REGION Network 7: flowrate ratio difference
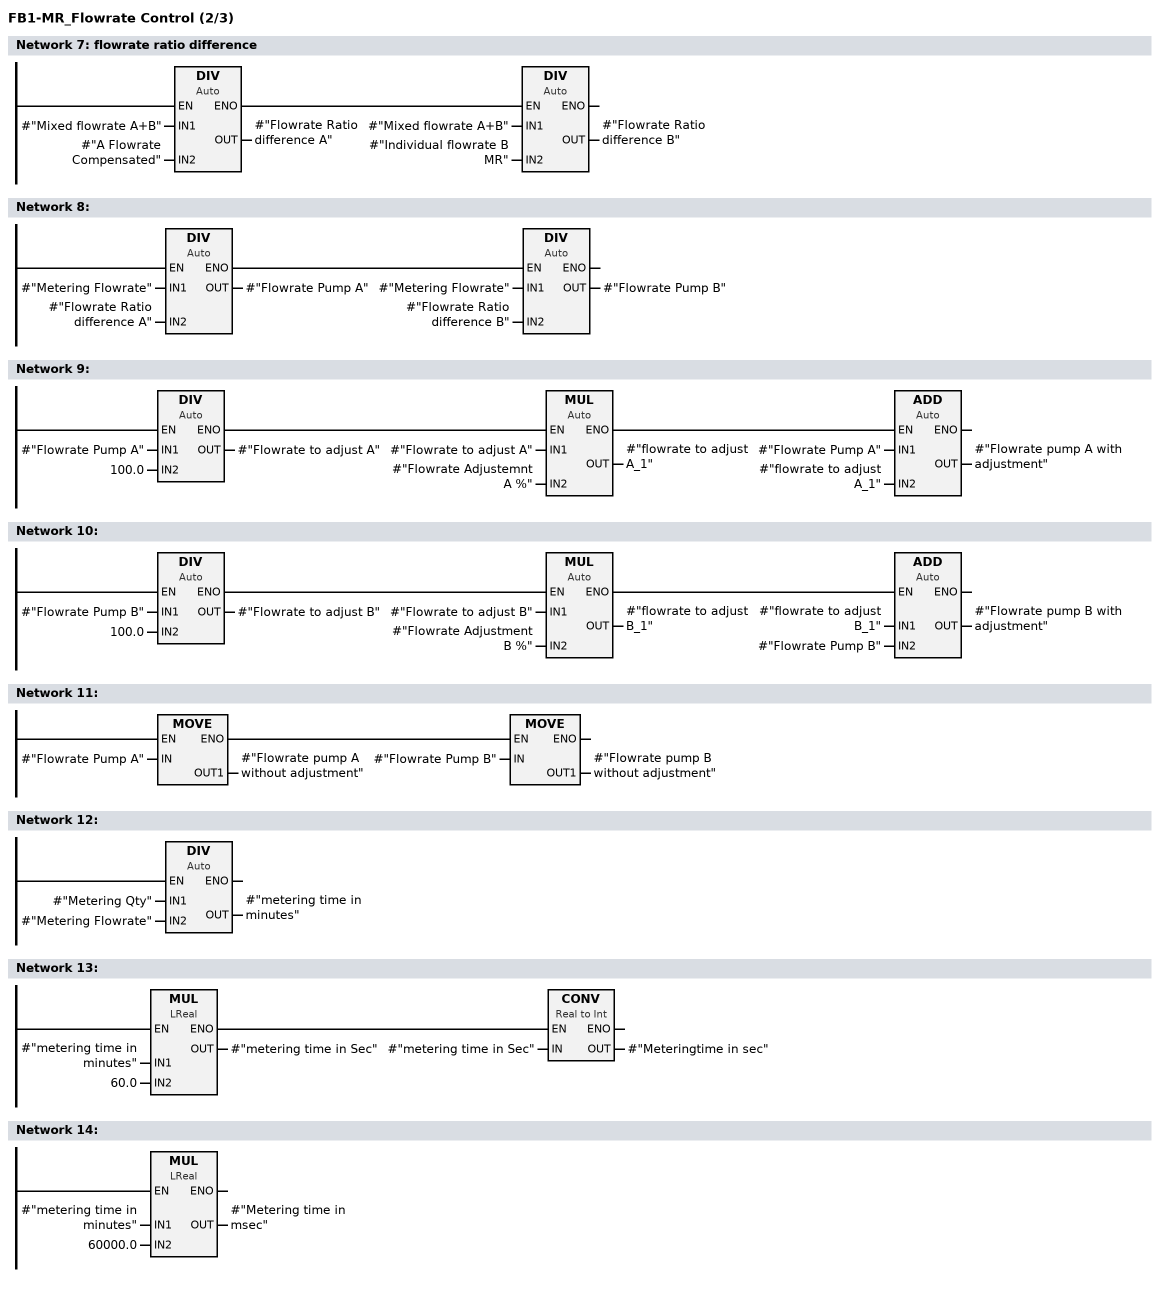
   RUNG wire#powerrail
      Div(in1 := #"Mixed flowrate A+B", in2 := #"A Flowrate Compensated", out => #"Flowrate Ratio difference A")
      Div(in1 := #"Mixed flowrate A+B", in2 := #"Individual flowrate B MR", out => #"Flowrate Ratio difference B")
   END_RUNG
   // the same network as SCL:
   #"Flowrate Ratio difference A" := #"Mixed flowrate A+B" / #"A Flowrate Compensated";
   #"Flowrate Ratio difference B" := #"Mixed flowrate A+B" / #"Individual flowrate B MR";
END_REGION

REGION Network 8
   RUNG wire#powerrail
      Div(in1 := #"Metering Flowrate", in2 := #"Flowrate Ratio difference A", out => #"Flowrate Pump A")
      Div(in1 := #"Metering Flowrate", in2 := #"Flowrate Ratio difference B", out => #"Flowrate Pump B")
   END_RUNG
   // the same network as SCL:
   #"Flowrate Pump A" := #"Metering Flowrate" / #"Flowrate Ratio difference A";
   #"Flowrate Pump B" := #"Metering Flowrate" / #"Flowrate Ratio difference B";
END_REGION

REGION Network 9
   RUNG wire#powerrail
      Div(in1 := #"Flowrate Pump A", in2 := 100.0, out => #"Flowrate to adjust A")
      Mul(in1 := #"Flowrate to adjust A", in2 := #"Flowrate Adjustemnt A %", out => #"flowrate to adjust A_1")
      Add(in1 := #"Flowrate Pump A", in2 := #"flowrate to adjust A_1", out => #"Flowrate pump A with adjustment")
   END_RUNG
   // the same network as SCL:
   #"Flowrate to adjust A" := #"Flowrate Pump A" / 100.0;
   #"flowrate to adjust A_1" := #"Flowrate to adjust A" * #"Flowrate Adjustemnt A %";
   #"Flowrate pump A with adjustment" := #"Flowrate Pump A" + #"flowrate to adjust A_1";
END_REGION

REGION Network 10
   RUNG wire#powerrail
      Div(in1 := #"Flowrate Pump B", in2 := 100.0, out => #"Flowrate to adjust B")
      Mul(in1 := #"Flowrate to adjust B", in2 := #"Flowrate Adjustment B %", out => #"flowrate to adjust B_1")
      Add(in1 := #"flowrate to adjust B_1", in2 := #"Flowrate Pump B", out => #"Flowrate pump B with adjustment")
   END_RUNG
   // the same network as SCL:
   #"Flowrate to adjust B" := #"Flowrate Pump B" / 100.0;
   #"flowrate to adjust B_1" := #"Flowrate to adjust B" * #"Flowrate Adjustment B %";
   #"Flowrate pump B with adjustment" := #"flowrate to adjust B_1" + #"Flowrate Pump B";
END_REGION

REGION Network 11
   RUNG wire#powerrail
      Move(in := #"Flowrate Pump A", out1 => #"Flowrate pump A without adjustment")
      Move(in := #"Flowrate Pump B", out1 => #"Flowrate pump B without adjustment")
   END_RUNG
   // the same network as SCL:
   #"Flowrate pump A without adjustment" := #"Flowrate Pump A";
   #"Flowrate pump B without adjustment" := #"Flowrate Pump B";
END_REGION

REGION Network 12
   RUNG wire#powerrail
      Div(in1 := #"Metering Qty", in2 := #"Metering Flowrate", out => #"metering time in minutes")
   END_RUNG
   // the same network as SCL:
   #"metering time in minutes" := #"Metering Qty" / #"Metering Flowrate";
END_REGION

REGION Network 13
   RUNG wire#powerrail
      { S7_Templates := "SrcType := LReal" } Mul(in1 := #"metering time in minutes", in2 := 60.0, out => #"metering time in Sec")
      { S7_Templates := "[SrcType := Real, DestType := Int]" } Convert(in := #"metering time in Sec", out => #"Meteringtime in sec")
   END_RUNG
   // the same network as SCL:
   #"metering time in Sec" := #"metering time in minutes" * 60.0;
   #"Meteringtime in sec" := REAL_TO_INT(#"metering time in Sec");
END_REGION

REGION Network 14
   RUNG wire#powerrail
      { S7_Templates := "SrcType := LReal" } Mul(in1 := #"metering time in minutes", in2 := 60000.0, out => #"Metering time in msec")
   END_RUNG
   // the same network as SCL:
   #"Metering time in msec" := #"metering time in minutes" * 60000.0;
END_REGION

REGION Network 15
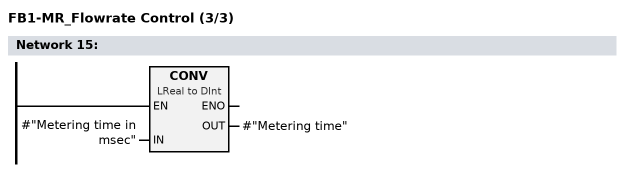
   RUNG wire#powerrail
      { S7_Templates := "[SrcType := LReal, DestType := DInt]" } Convert(in := #"Metering time in msec", out => #"Metering time")
   END_RUNG
   // the same network as SCL:
   #"Metering time" := LREAL_TO_DINT(#"Metering time in msec");
END_REGION
END_FUNCTION_BLOCK

ORGANIZATION_BLOCK "Startup"   // OB100, LAD, Startup
TITLE = "Complete Restart"
{ S7_Optimized_Access := 'TRUE' }
VERSION : 0.1
// stored: AutoNumber true, IsIECCheckEnabled false, SetENOAutomatically false
   VAR_INPUT
      LostRetentive : Bool;   // True if retentive data are lost
      LostRTC : Bool;   // True if date and time are lost
   END_VAR
BEGIN

REGION Network 1
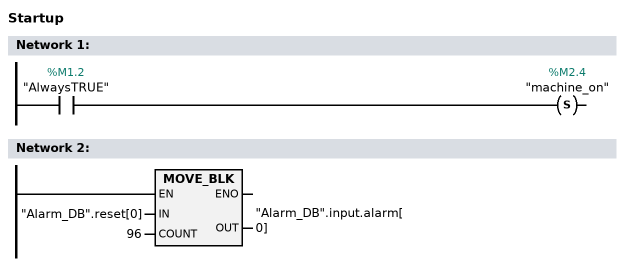
   RUNG wire#powerrail
      Contact( "AlwaysTRUE" )
      S_Coil( "machine_on" )
   END_RUNG
   // the same network as SCL:
   IF "AlwaysTRUE" THEN "machine_on" := TRUE; END_IF;
END_REGION

REGION Network 2
   MOVE_BLK(IN := "Alarm_DB".reset[0], COUNT := 96, OUT => "Alarm_DB".input.alarm[0]);
END_REGION
END_ORGANIZATION_BLOCK

FUNCTION "Alram_Scroll" : Void   // FC15, LAD
{ S7_Optimized_Access := 'TRUE' }
VERSION : 0.1
// stored: AutoNumber true, IsIECCheckEnabled false, SetENOAutomatically false, UDAEnableTagReadback false
   VAR CONSTANT
      "AlramDisplay time" : DInt := 2000;
   END_VAR
BEGIN

REGION Network 1
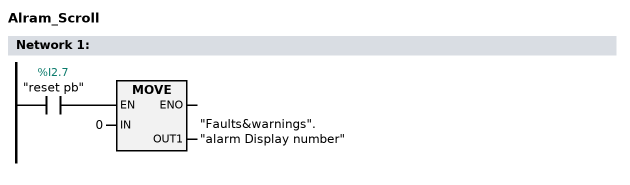
   RUNG wire#powerrail
      Contact( "reset pb" )
      Move(in := 0, out1 => "Faults&warnings"."alarm Display number")
   END_RUNG
   // the same network as SCL:
   IF "reset pb" THEN "Faults&warnings"."alarm Display number" := 0; END_IF;
END_REGION
END_FUNCTION

FUNCTION_BLOCK "FB10-Condition Check"   // FB10, LAD
{ S7_Optimized_Access := 'TRUE' }
VERSION : 0.1
// stored: AutoNumber false, IsIECCheckEnabled false, IsRetainMemResEnabled false, MemoryReserve 100, SetENOAutomatically false, UDAEnableTagReadback false
   VAR_INPUT
      "Time" : DInt;
      "Pump ON delay" : DInt;
      Check_Time { ExternalAccessible := 'False'; ExternalVisible := 'False'; ExternalWritable := 'False'} : DInt;
      Pressure_SP { ExternalAccessible := 'False'; ExternalVisible := 'False'; ExternalWritable := 'False'} : Real;
      Pressure_tolerance { ExternalAccessible := 'False'; ExternalVisible := 'False'; ExternalWritable := 'False'} : Real;
      Current_pressure { ExternalAccessible := 'False'; ExternalVisible := 'False'; ExternalWritable := 'False'} : Real;
      selected { ExternalAccessible := 'False'; ExternalVisible := 'False'; ExternalWritable := 'False'} : Bool;
   END_VAR
   VAR_OUTPUT
      "dispensing Time PV" : Int;
      "Checking Time pv" { ExternalAccessible := 'False'; ExternalVisible := 'False'; ExternalWritable := 'False'} : Int;
      test_ok { ExternalAccessible := 'False'; ExternalVisible := 'False'; ExternalWritable := 'False'} : Bool;
      test_nok { ExternalAccessible := 'False'; ExternalVisible := 'False'; ExternalWritable := 'False'} : Bool;
      test_fail { ExternalAccessible := 'False'; ExternalVisible := 'False'; ExternalWritable := 'False'} : Bool;
   END_VAR
   VAR_IN_OUT
      "Start ConditonCheck" : Bool;
      "Stop ConditonCheck" : Bool;
      "ConditonCheck Running" : Bool;
      "ConditonCheck completed" : Bool;
      "ON Gear Pump" : Bool;
      "ON inlet" : Bool;
   END_VAR
   VAR
      "dispensing time done" : Bool;
      "dispensing time in sec" : DInt;
      "timer in sec" : DInt;
      "timer PV in sec" : DInt;
      "timer input" : DInt;
      IEC_Timer_0_Instance { S7_SetPoint := 'True'} : TON_TIME;
      IEC_Timer_0_Instance_1 { S7_SetPoint := 'True'} : TON_TIME;
      IEC_Timer_0_Instance_2 { S7_SetPoint := 'True'} : TON_TIME;
      IEC_Timer_0_Instance_4 { S7_SetPoint := 'True'} : TON_TIME;
      "Press+ve" { ExternalAccessible := 'False'; ExternalVisible := 'False'; ExternalWritable := 'False'; S7_SetPoint := 'True'} : Real;
      "Press-ve" { ExternalAccessible := 'False'; ExternalVisible := 'False'; ExternalWritable := 'False'} : Real;
      IEC_Timer_0_Instance_3 { ExternalAccessible := 'False'; ExternalVisible := 'False'; ExternalWritable := 'False'; S7_SetPoint := 'True'} : TON_TIME;
      Checktime_ms { ExternalAccessible := 'False'; ExternalVisible := 'False'; ExternalWritable := 'False'; S7_SetPoint := 'True'} : DInt;
      Check_timesec { ExternalAccessible := 'False'; ExternalVisible := 'False'; ExternalWritable := 'False'} : DInt;
      temp_ons { ExternalAccessible := 'False'; ExternalVisible := 'False'; ExternalWritable := 'False'} : Bool;
   END_VAR
   VAR_TEMP   // added for the SCL form of the ladder/FBD networks
      _w1 : Bool;
   END_VAR
BEGIN

REGION Network 1
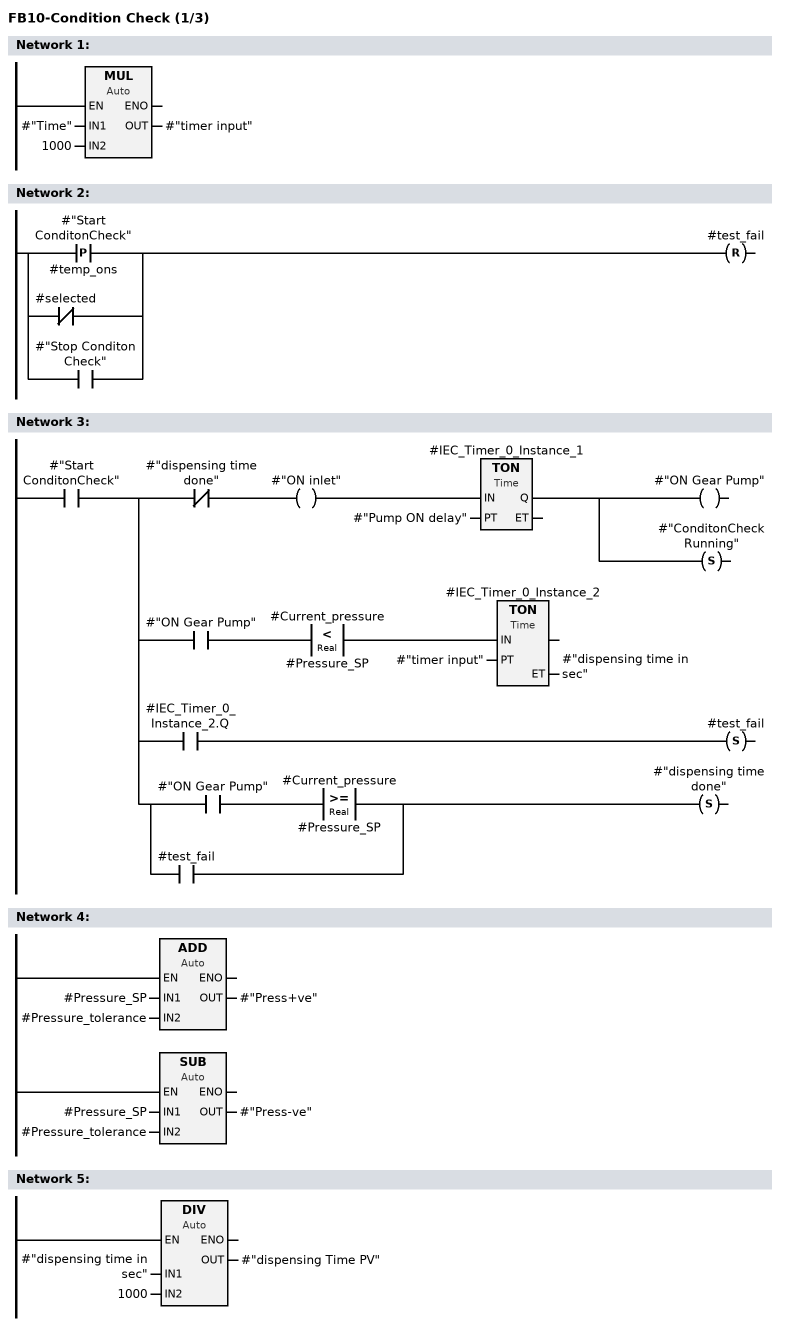
   RUNG wire#powerrail
      Mul(in1 := #"Time", in2 := 1000, out => #"timer input")
   END_RUNG
   // the same network as SCL:
   #"timer input" := #"Time" * 1000;
END_REGION

REGION Network 2
   RUNG wire#powerrail
      P_Contact(operand := #"Start ConditonCheck", bit := #temp_ons)
      wire#w1
      R_Coil( #test_fail )
   END_RUNG
   RUNG wire#powerrail
      I_Contact( #selected )
   END_RUNG wire#w1
   RUNG wire#powerrail
      Contact( #"Stop ConditonCheck" )
   END_RUNG wire#w1
   // the same network as SCL:
   #_w1 := #"Start ConditonCheck" AND NOT #temp_ons;   // rising edge of #"Start ConditonCheck"
   #temp_ons := #"Start ConditonCheck";
   IF #_w1 OR NOT #selected OR #"Stop ConditonCheck" THEN #test_fail := FALSE; END_IF;
END_REGION

REGION Network 3
   RUNG wire#powerrail
      Contact( #"Start ConditonCheck" )
      wire#w1
      I_Contact( #"dispensing time done" )
      Coil( #"ON inlet" )
      { S7_Templates := "time_type := Time" } #IEC_Timer_0_Instance_1.TON(pt := #"Pump ON delay", et =>)
      wire#w2
      Coil( #"ON Gear Pump" )
   END_RUNG
   RUNG wire#w2
      S_Coil( #"ConditonCheck Running" )
   END_RUNG
   RUNG wire#w1
      Contact( #"ON Gear Pump" )
      { S7_Templates := "SrcType := Real" } LT_Contact(in1 := #Current_pressure, in2 := #Pressure_SP)
      { S7_Templates := "time_type := Time" } #IEC_Timer_0_Instance_2.TON(pt := #"timer input", et => #"dispensing time in sec")
   END_RUNG
   RUNG wire#w1
      Contact( #IEC_Timer_0_Instance_2.Q )
      S_Coil( #test_fail )
   END_RUNG
   RUNG wire#w1
      Contact( #"ON Gear Pump" )
      { S7_Templates := "SrcType := Real" } GE_Contact(in1 := #Current_pressure, in2 := #Pressure_SP)
      wire#w3
      S_Coil( #"dispensing time done" )
   END_RUNG
   RUNG wire#w1
      Contact( #test_fail )
   END_RUNG wire#w3
   // the same network as SCL:
   #"ON inlet" := #"Start ConditonCheck" AND NOT #"dispensing time done";
   #IEC_Timer_0_Instance_1(IN := #"ON inlet", PT := #"Pump ON delay");   // TON
   #"ON Gear Pump" := #IEC_Timer_0_Instance_1.Q;
   IF #IEC_Timer_0_Instance_1.Q THEN #"ConditonCheck Running" := TRUE; END_IF;
   #IEC_Timer_0_Instance_2(IN := #"Start ConditonCheck" AND #"ON Gear Pump" AND (#Current_pressure < #Pressure_SP),   // TON
                           PT := #"timer input",
                           ET => #"dispensing time in sec");
   IF #"Start ConditonCheck" AND #IEC_Timer_0_Instance_2.Q THEN #test_fail := TRUE; END_IF;
   IF #"Start ConditonCheck" AND ((#"ON Gear Pump" AND (#Current_pressure >= #Pressure_SP)) OR #test_fail) THEN
       #"dispensing time done" := TRUE;
   END_IF;
END_REGION

REGION Network 4
   RUNG wire#powerrail
      Add(in1 := #Pressure_SP, in2 := #Pressure_tolerance, out => #"Press+ve")
   END_RUNG
   RUNG wire#powerrail
      Sub(in1 := #Pressure_SP, in2 := #Pressure_tolerance, out => #"Press-ve")
   END_RUNG
   // the same network as SCL:
   #"Press+ve" := #Pressure_SP + #Pressure_tolerance;
   #"Press-ve" := #Pressure_SP - #Pressure_tolerance;
END_REGION

REGION Network 5
   RUNG wire#powerrail
      Div(in1 := #"dispensing time in sec", in2 := 1000, out => #"dispensing Time PV")
   END_RUNG
   // the same network as SCL:
   #"dispensing Time PV" := #"dispensing time in sec" / 1000;
END_REGION

REGION Network 6
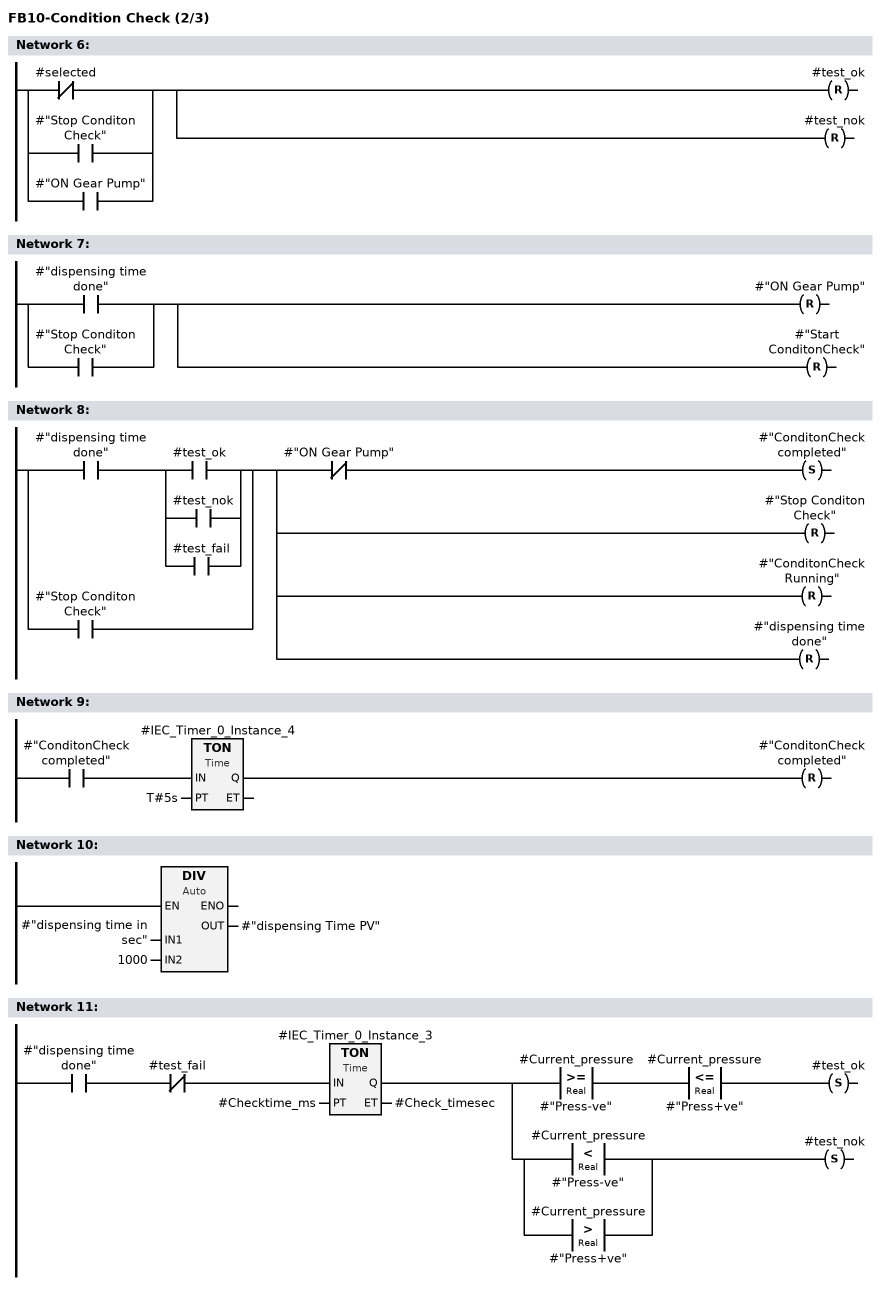
   RUNG wire#powerrail
      I_Contact( #selected )
      wire#w1
      R_Coil( #test_ok )
   END_RUNG
   RUNG wire#powerrail
      Contact( #"Stop ConditonCheck" )
   END_RUNG wire#w1
   RUNG wire#powerrail
      Contact( #"ON Gear Pump" )
   END_RUNG wire#w1
   RUNG wire#w1
      R_Coil( #test_nok )
   END_RUNG
   // the same network as SCL:
   IF NOT #selected OR #"Stop ConditonCheck" OR #"ON Gear Pump" THEN
       #test_ok := FALSE;
       #test_nok := FALSE;
   END_IF;
END_REGION

REGION Network 7
   RUNG wire#powerrail
      Contact( #"dispensing time done" )
      wire#w1
      R_Coil( #"ON Gear Pump" )
   END_RUNG
   RUNG wire#powerrail
      Contact( #"Stop ConditonCheck" )
   END_RUNG wire#w1
   RUNG wire#w1
      R_Coil( #"Start ConditonCheck" )
   END_RUNG
   // the same network as SCL:
   IF #"dispensing time done" OR #"Stop ConditonCheck" THEN
       #"ON Gear Pump" := FALSE;
       #"Start ConditonCheck" := FALSE;
   END_IF;
END_REGION

REGION Network 8
   RUNG wire#powerrail
      Contact( #"dispensing time done" )
      wire#w1
      Contact( #test_ok )
      wire#w2
      I_Contact( #"ON Gear Pump" )
      S_Coil( #"ConditonCheck completed" )
   END_RUNG
   RUNG wire#w1
      Contact( #test_nok )
   END_RUNG wire#w2
   RUNG wire#w1
      Contact( #test_fail )
   END_RUNG wire#w2
   RUNG wire#powerrail
      Contact( #"Stop ConditonCheck" )
   END_RUNG wire#w2
   RUNG wire#w2
      R_Coil( #"Stop ConditonCheck" )
   END_RUNG
   RUNG wire#w2
      R_Coil( #"ConditonCheck Running" )
   END_RUNG
   RUNG wire#w2
      R_Coil( #"dispensing time done" )
   END_RUNG
   // the same network as SCL:
   #_w1 := (#"dispensing time done" AND (#test_ok OR #test_nok OR #test_fail)) OR #"Stop ConditonCheck";
   IF #_w1 AND NOT #"ON Gear Pump" THEN #"ConditonCheck completed" := TRUE; END_IF;
   IF #_w1 THEN
       #"Stop ConditonCheck" := FALSE;
       #"ConditonCheck Running" := FALSE;
       #"dispensing time done" := FALSE;
   END_IF;
END_REGION

REGION Network 9
   RUNG wire#powerrail
      Contact( #"ConditonCheck completed" )
      { S7_Templates := "time_type := Time" } #IEC_Timer_0_Instance_4.TON(pt := T#5s, et =>)
      R_Coil( #"ConditonCheck completed" )
   END_RUNG
   // the same network as SCL:
   #IEC_Timer_0_Instance_4(IN := #"ConditonCheck completed", PT := T#5s);   // TON
   IF #IEC_Timer_0_Instance_4.Q THEN #"ConditonCheck completed" := FALSE; END_IF;
END_REGION

REGION Network 10
   RUNG wire#powerrail
      Div(in1 := #"dispensing time in sec", in2 := 1000, out => #"dispensing Time PV")
   END_RUNG
   // the same network as SCL:
   #"dispensing Time PV" := #"dispensing time in sec" / 1000;
END_REGION

REGION Network 11
   RUNG wire#powerrail
      Contact( #"dispensing time done" )
      I_Contact( #test_fail )
      { S7_Templates := "time_type := Time" } #IEC_Timer_0_Instance_3.TON(pt := #Checktime_ms, et => #Check_timesec)
      wire#w1
      { S7_Templates := "SrcType := Real" } GE_Contact(in1 := #Current_pressure, in2 := #"Press-ve")
      { S7_Templates := "SrcType := Real" } LE_Contact(in1 := #Current_pressure, in2 := #"Press+ve")
      S_Coil( #test_ok )
   END_RUNG
   RUNG wire#w1
      { S7_Templates := "SrcType := Real" } LT_Contact(in1 := #Current_pressure, in2 := #"Press-ve")
      wire#w2
      S_Coil( #test_nok )
   END_RUNG
   RUNG wire#w1
      { S7_Templates := "SrcType := Real" } GT_Contact(in1 := #Current_pressure, in2 := #"Press+ve")
   END_RUNG wire#w2
   // the same network as SCL:
   #IEC_Timer_0_Instance_3(IN := #"dispensing time done" AND NOT #test_fail,   // TON
                           PT := #Checktime_ms,
                           ET => #Check_timesec);
   IF #IEC_Timer_0_Instance_3.Q AND (#Current_pressure >= #"Press-ve") AND (#Current_pressure <= #"Press+ve") THEN
       #test_ok := TRUE;
   END_IF;
   IF #IEC_Timer_0_Instance_3.Q AND ((#Current_pressure < #"Press-ve") OR (#Current_pressure > #"Press+ve")) THEN
       #test_nok := TRUE;
   END_IF;
END_REGION

REGION Network 12
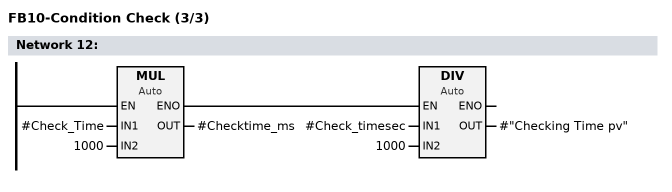
   RUNG wire#powerrail
      Mul(in1 := #Check_Time, in2 := 1000, out => #Checktime_ms)
      Div(in1 := #Check_timesec, in2 := 1000, out => #"Checking Time pv")
   END_RUNG
   // the same network as SCL:
   #Checktime_ms := #Check_Time * 1000;
   #"Checking Time pv" := #Check_timesec / 1000;
END_REGION
END_FUNCTION_BLOCK

FUNCTION_BLOCK "MixingRatio"   // FB11, LAD
{ S7_Optimized_Access := 'TRUE' }
VERSION : 0.1
// stored: AutoNumber true, IsIECCheckEnabled false, IsRetainMemResEnabled false, MemoryReserve 100, SetENOAutomatically false, UDAEnableTagReadback false
   VAR_INPUT
      "Pump size A in ml" : Real;
      "Pump size B in ml" : Real;
      "Pump speed A_Max" : Real;
      "Pump speed B_Max" : Real;
      "Pump speed A_Passive" : Real;
      "Pump speed B_Passive" : Real;
      "Mixing ratio A100:B" : Real;
      "No.of Component" : Int;
      "Density A" : Real;
      "Density B" : Real;
      "Mixed Flowrate Set" : Real;
      "Flowrate Type" : Int;
   END_VAR
   VAR_OUTPUT
      "Maximum Flowrate A" : Real;
      "Maximum Flowrate B" : Real;
      "Maximum Flowrate A_Limited" : Real;
      "Maximum Flowrate B_Limited" : Real;
      "Maximum Flowrate Mixed" : Real;
      "Required flowrate A" : Real;
      "Required flowrate B" : Real;
   END_VAR
   VAR
      "Pump size A actual" : Real;
      "Pump size B actual" : Real;
      "Max flowrate A" : Real;
      "Max flowrate B" : Real;
      "Ratio margin B" : Real;
      "usable A flowrate per B ratio" : Real;
      "maximum mixed flowrate" : Real;
      "usable flowrate A per ratio" : Real;
      "usable flowrate B per ratio" : Real;
      "Flowrate difference A" : Real;
      "Flowrate difference B" : Real;
      "target flowrate A" : Real;
      "target flowrate B" : Real;
   END_VAR
   VAR_TEMP   // added for the SCL form of the ladder/FBD networks
      _w1 : Bool;
   END_VAR
BEGIN

REGION Network 1
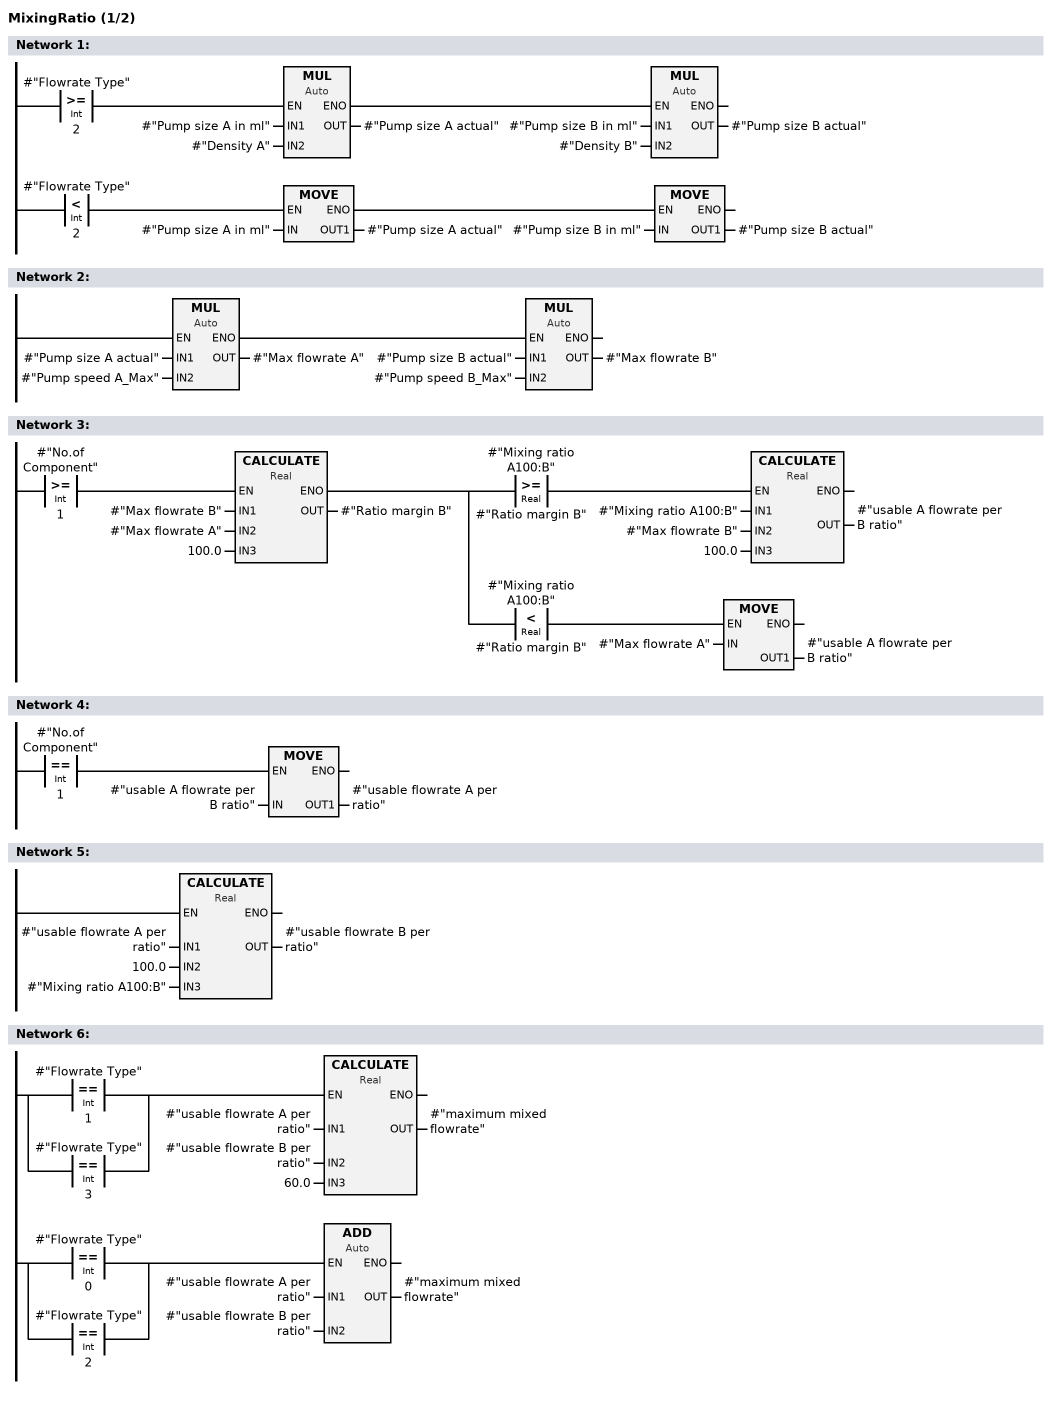
   RUNG wire#powerrail
      { S7_Templates := "SrcType := Int" } GE_Contact(in1 := #"Flowrate Type", in2 := 2)
      Mul(in1 := #"Pump size A in ml", in2 := #"Density A", out => #"Pump size A actual")
      Mul(in1 := #"Pump size B in ml", in2 := #"Density B", out => #"Pump size B actual")
   END_RUNG
   RUNG wire#powerrail
      { S7_Templates := "SrcType := Int" } LT_Contact(in1 := #"Flowrate Type", in2 := 2)
      Move(in := #"Pump size A in ml", out1 => #"Pump size A actual")
      Move(in := #"Pump size B in ml", out1 => #"Pump size B actual")
   END_RUNG
   // the same network as SCL:
   IF #"Flowrate Type" >= 2 THEN
       #"Pump size A actual" := #"Pump size A in ml" * #"Density A";
       #"Pump size B actual" := #"Pump size B in ml" * #"Density B";
   END_IF;
   IF #"Flowrate Type" < 2 THEN
       #"Pump size A actual" := #"Pump size A in ml";
       #"Pump size B actual" := #"Pump size B in ml";
   END_IF;
END_REGION

REGION Network 2
   RUNG wire#powerrail
      Mul(in1 := #"Pump size A actual", in2 := #"Pump speed A_Max", out => #"Max flowrate A")
      Mul(in1 := #"Pump size B actual", in2 := #"Pump speed B_Max", out => #"Max flowrate B")
   END_RUNG
   // the same network as SCL:
   #"Max flowrate A" := #"Pump size A actual" * #"Pump speed A_Max";
   #"Max flowrate B" := #"Pump size B actual" * #"Pump speed B_Max";
END_REGION

REGION Network 3
   RUNG wire#powerrail
      { S7_Templates := "SrcType := Int" } GE_Contact(in1 := #"No.of Component", in2 := 1)
      { S7_Templates := "SrcType := Real"; S7_Expression := "(IN1/IN2)*IN3" } Calculate(in1 := #"Max flowrate B", in2 := #"Max flowrate A", in3 := 100.0, out => #"Ratio margin B")
      wire#w1
      { S7_Templates := "SrcType := Real" } GE_Contact(in1 := #"Mixing ratio A100:B", in2 := #"Ratio margin B")
      { S7_Templates := "SrcType := Real"; S7_Expression := "IN2/(IN1/IN3)" } Calculate(in1 := #"Mixing ratio A100:B", in2 := #"Max flowrate B", in3 := 100.0, out => #"usable A flowrate per B ratio")
   END_RUNG
   RUNG wire#w1
      { S7_Templates := "SrcType := Real" } LT_Contact(in1 := #"Mixing ratio A100:B", in2 := #"Ratio margin B")
      Move(in := #"Max flowrate A", out1 => #"usable A flowrate per B ratio")
   END_RUNG
   // the same network as SCL:
   #_w1 := #"No.of Component" >= 1;
   IF #_w1 THEN #"Ratio margin B" := (#"Max flowrate B"/#"Max flowrate A")*100.0; END_IF;
   IF #_w1 AND (#"Mixing ratio A100:B" >= #"Ratio margin B") THEN
       #"usable A flowrate per B ratio" := #"Max flowrate B"/(#"Mixing ratio A100:B"/100.0);
   END_IF;
   IF #_w1 AND (#"Mixing ratio A100:B" < #"Ratio margin B") THEN
       #"usable A flowrate per B ratio" := #"Max flowrate A";
   END_IF;
END_REGION

REGION Network 4
   RUNG wire#powerrail
      { S7_Templates := "SrcType := Int" } EQ_Contact(in1 := #"No.of Component", in2 := 1)
      Move(in := #"usable A flowrate per B ratio", out1 => #"usable flowrate A per ratio")
   END_RUNG
   // the same network as SCL:
   IF #"No.of Component" = 1 THEN #"usable flowrate A per ratio" := #"usable A flowrate per B ratio"; END_IF;
END_REGION

REGION Network 5
   RUNG wire#powerrail
      { S7_Templates := "SrcType := Real"; S7_Expression := "(IN1/IN2)*IN3" } Calculate(in1 := #"usable flowrate A per ratio", in2 := 100.0, in3 := #"Mixing ratio A100:B", out => #"usable flowrate B per ratio")
   END_RUNG
   // the same network as SCL:
   #"usable flowrate B per ratio" := (#"usable flowrate A per ratio"/100.0)*#"Mixing ratio A100:B";
END_REGION

REGION Network 6
   RUNG wire#powerrail
      { S7_Templates := "SrcType := Int" } EQ_Contact(in1 := #"Flowrate Type", in2 := 1)
      wire#w1
      { S7_Templates := "SrcType := Real"; S7_Expression := "(IN1+IN2)/IN3" } Calculate(in1 := #"usable flowrate A per ratio", in2 := #"usable flowrate B per ratio", in3 := 60.0, out => #"maximum mixed flowrate")
   END_RUNG
   RUNG wire#powerrail
      { S7_Templates := "SrcType := Int" } EQ_Contact(in1 := #"Flowrate Type", in2 := 3)
   END_RUNG wire#w1
   RUNG wire#powerrail
      { S7_Templates := "SrcType := Int" } EQ_Contact(in1 := #"Flowrate Type", in2 := 0)
      wire#w2
      Add(in1 := #"usable flowrate A per ratio", in2 := #"usable flowrate B per ratio", out => #"maximum mixed flowrate")
   END_RUNG
   RUNG wire#powerrail
      { S7_Templates := "SrcType := Int" } EQ_Contact(in1 := #"Flowrate Type", in2 := 2)
   END_RUNG wire#w2
   // the same network as SCL:
   IF (#"Flowrate Type" = 1) OR (#"Flowrate Type" = 3) THEN
       #"maximum mixed flowrate" := (#"usable flowrate A per ratio"+#"usable flowrate B per ratio")/60.0;
   END_IF;
   IF (#"Flowrate Type" = 0) OR (#"Flowrate Type" = 2) THEN
       #"maximum mixed flowrate" := #"usable flowrate A per ratio" + #"usable flowrate B per ratio";
   END_IF;
END_REGION

REGION Network 7
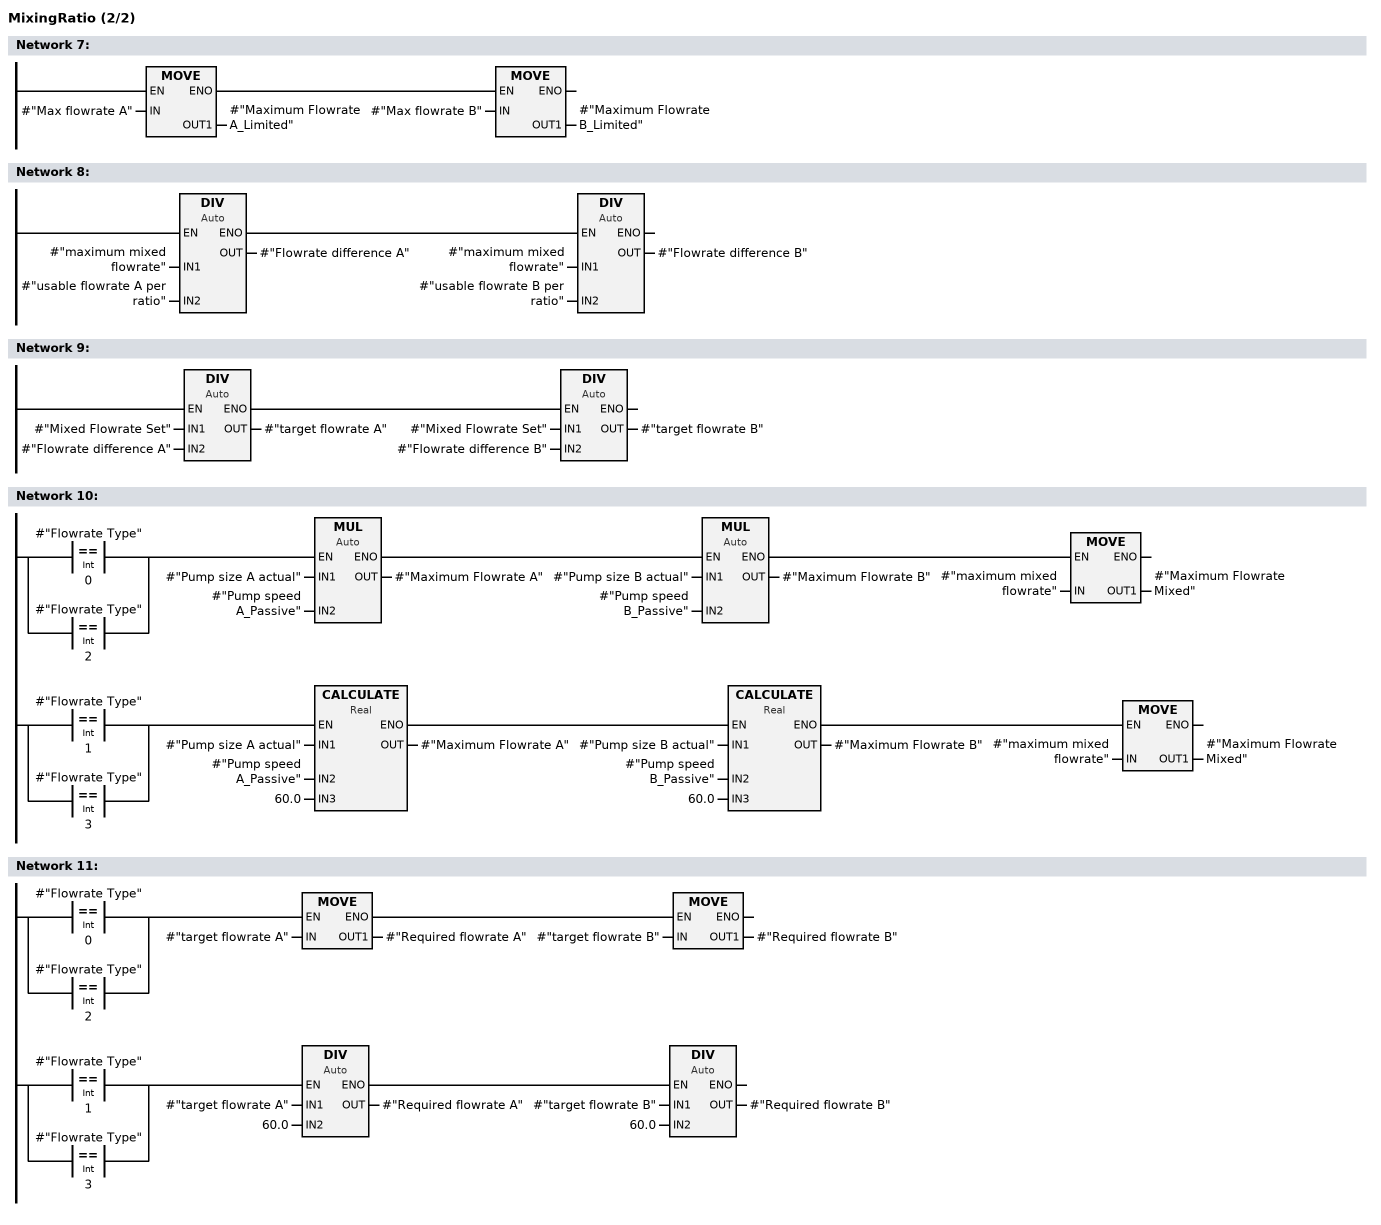
   RUNG wire#powerrail
      Move(in := #"Max flowrate A", out1 => #"Maximum Flowrate A_Limited")
      Move(in := #"Max flowrate B", out1 => #"Maximum Flowrate B_Limited")
   END_RUNG
   // the same network as SCL:
   #"Maximum Flowrate A_Limited" := #"Max flowrate A";
   #"Maximum Flowrate B_Limited" := #"Max flowrate B";
END_REGION

REGION Network 8
   RUNG wire#powerrail
      Div(in1 := #"maximum mixed flowrate", in2 := #"usable flowrate A per ratio", out => #"Flowrate difference A")
      Div(in1 := #"maximum mixed flowrate", in2 := #"usable flowrate B per ratio", out => #"Flowrate difference B")
   END_RUNG
   // the same network as SCL:
   #"Flowrate difference A" := #"maximum mixed flowrate" / #"usable flowrate A per ratio";
   #"Flowrate difference B" := #"maximum mixed flowrate" / #"usable flowrate B per ratio";
END_REGION

REGION Network 9
   RUNG wire#powerrail
      Div(in1 := #"Mixed Flowrate Set", in2 := #"Flowrate difference A", out => #"target flowrate A")
      Div(in1 := #"Mixed Flowrate Set", in2 := #"Flowrate difference B", out => #"target flowrate B")
   END_RUNG
   // the same network as SCL:
   #"target flowrate A" := #"Mixed Flowrate Set" / #"Flowrate difference A";
   #"target flowrate B" := #"Mixed Flowrate Set" / #"Flowrate difference B";
END_REGION

REGION Network 10
   RUNG wire#powerrail
      { S7_Templates := "SrcType := Int" } EQ_Contact(in1 := #"Flowrate Type", in2 := 0)
      wire#w1
      Mul(in1 := #"Pump size A actual", in2 := #"Pump speed A_Passive", out => #"Maximum Flowrate A")
      Mul(in1 := #"Pump size B actual", in2 := #"Pump speed B_Passive", out => #"Maximum Flowrate B")
      Move(in := #"maximum mixed flowrate", out1 => #"Maximum Flowrate Mixed")
   END_RUNG
   RUNG wire#powerrail
      { S7_Templates := "SrcType := Int" } EQ_Contact(in1 := #"Flowrate Type", in2 := 2)
   END_RUNG wire#w1
   RUNG wire#powerrail
      { S7_Templates := "SrcType := Int" } EQ_Contact(in1 := #"Flowrate Type", in2 := 1)
      wire#w2
      { S7_Templates := "SrcType := Real"; S7_Expression := "(IN1*IN2)/IN3" } Calculate(in1 := #"Pump size A actual", in2 := #"Pump speed A_Passive", in3 := 60.0, out => #"Maximum Flowrate A")
      { S7_Templates := "SrcType := Real"; S7_Expression := "(IN1*IN2)/IN3" } Calculate(in1 := #"Pump size B actual", in2 := #"Pump speed B_Passive", in3 := 60.0, out => #"Maximum Flowrate B")
      Move(in := #"maximum mixed flowrate", out1 => #"Maximum Flowrate Mixed")
   END_RUNG
   RUNG wire#powerrail
      { S7_Templates := "SrcType := Int" } EQ_Contact(in1 := #"Flowrate Type", in2 := 3)
   END_RUNG wire#w2
   // the same network as SCL:
   IF (#"Flowrate Type" = 0) OR (#"Flowrate Type" = 2) THEN
       #"Maximum Flowrate A" := #"Pump size A actual" * #"Pump speed A_Passive";
       #"Maximum Flowrate B" := #"Pump size B actual" * #"Pump speed B_Passive";
       #"Maximum Flowrate Mixed" := #"maximum mixed flowrate";
   END_IF;
   IF (#"Flowrate Type" = 1) OR (#"Flowrate Type" = 3) THEN
       #"Maximum Flowrate A" := (#"Pump size A actual"*#"Pump speed A_Passive")/60.0;
       #"Maximum Flowrate B" := (#"Pump size B actual"*#"Pump speed B_Passive")/60.0;
       #"Maximum Flowrate Mixed" := #"maximum mixed flowrate";
   END_IF;
END_REGION

REGION Network 11
   RUNG wire#powerrail
      { S7_Templates := "SrcType := Int" } EQ_Contact(in1 := #"Flowrate Type", in2 := 0)
      wire#w1
      Move(in := #"target flowrate A", out1 => #"Required flowrate A")
      Move(in := #"target flowrate B", out1 => #"Required flowrate B")
   END_RUNG
   RUNG wire#powerrail
      { S7_Templates := "SrcType := Int" } EQ_Contact(in1 := #"Flowrate Type", in2 := 2)
   END_RUNG wire#w1
   RUNG wire#powerrail
      { S7_Templates := "SrcType := Int" } EQ_Contact(in1 := #"Flowrate Type", in2 := 1)
      wire#w2
      Div(in1 := #"target flowrate A", in2 := 60.0, out => #"Required flowrate A")
      Div(in1 := #"target flowrate B", in2 := 60.0, out => #"Required flowrate B")
   END_RUNG
   RUNG wire#powerrail
      { S7_Templates := "SrcType := Int" } EQ_Contact(in1 := #"Flowrate Type", in2 := 3)
   END_RUNG wire#w2
   // the same network as SCL:
   IF (#"Flowrate Type" = 0) OR (#"Flowrate Type" = 2) THEN
       #"Required flowrate A" := #"target flowrate A";
       #"Required flowrate B" := #"target flowrate B";
   END_IF;
   IF (#"Flowrate Type" = 1) OR (#"Flowrate Type" = 3) THEN
       #"Required flowrate A" := #"target flowrate A" / 60.0;
       #"Required flowrate B" := #"target flowrate B" / 60.0;
   END_IF;
END_REGION
END_FUNCTION_BLOCK

FUNCTION "selection_Machine" : Void   // FC1, LAD
{ S7_Optimized_Access := 'TRUE' }
VERSION : 0.1
// stored: AutoNumber true, IsIECCheckEnabled false, SetENOAutomatically false, UDAEnableTagReadback false
BEGIN

REGION Network 1 (SCL)
   IF "selection_machie_db"."1k_2k" = TRUE THEN
       "Mixing ratio"."Mixing ratio set" := 0;
   END_IF;
END_REGION
END_FUNCTION

DATA_BLOCK "FB0-MR_Quantity Control_1_DB"   // DB24
VERSION : 0.1
// stored: AutoNumber true, DBAccessibleFromOPCUA true, InstanceOfName FB0-MR_Quantity Control_1, InstanceOfType FB
"FB0-MR_Quantity Control_1"
BEGIN
END_DATA_BLOCK

DATA_BLOCK "FB1-MR_Flowrate Control_DB"   // DB39
VERSION : 0.1
// stored: AutoNumber true, DBAccessibleFromOPCUA true, InstanceOfName FB1-MR_Flowrate Control, InstanceOfType FB
"FB1-MR_Flowrate Control"
BEGIN
END_DATA_BLOCK

DATA_BLOCK "FB10-Condition CheckA_DB"   // DB134
VERSION : 0.1
// stored: AutoNumber true, DBAccessibleFromOPCUA true, InstanceOfName FB10-Condition Check, InstanceOfType FB
"FB10-Condition Check"
BEGIN
END_DATA_BLOCK

DATA_BLOCK "FB10-Condition CheckB_DB"   // DB225
VERSION : 0.1
// stored: AutoNumber true, DBAccessibleFromOPCUA true, InstanceOfName FB10-Condition Check, InstanceOfType FB
"FB10-Condition Check"
BEGIN
END_DATA_BLOCK

DATA_BLOCK "FB10-Condition Check_1_DB"   // DB283
VERSION : 0.1
// stored: AutoNumber true, DBAccessibleFromOPCUA true, InstanceOfName FB10-Condition Check_1, InstanceOfType FB
"FB10-Condition Check_1"
BEGIN
END_DATA_BLOCK

DATA_BLOCK "FB10-Condition Check_1_DB_1"   // DB289
VERSION : 0.1
// stored: AutoNumber true, DBAccessibleFromOPCUA true, InstanceOfName FB10-Condition Check_1, InstanceOfType FB
"FB10-Condition Check_1"
BEGIN
END_DATA_BLOCK

DATA_BLOCK "FB2-meteringpgmFB_DB"   // DB59
VERSION : 0.1
// stored: AutoNumber true, DBAccessibleFromOPCUA true, InstanceOfName FB2-meteringFB, InstanceOfType FB
"FB2-meteringFB"
BEGIN
END_DATA_BLOCK

DATA_BLOCK "FB21-Flush A_DB"   // DB155
VERSION : 0.1
// stored: AutoNumber true, DBAccessibleFromOPCUA true, InstanceOfName FB21-Flush A, InstanceOfType FB
"FB21-Flush A"
BEGIN
END_DATA_BLOCK

DATA_BLOCK "FB21-Flush A_DB_1"   // DB160
VERSION : 0.1
// stored: AutoNumber true, DBAccessibleFromOPCUA true, InstanceOfName FB21-Flush A, InstanceOfType FB
"FB21-Flush A"
BEGIN
END_DATA_BLOCK

DATA_BLOCK "FB21-Flush A_DB_2"   // DB7
VERSION : 0.1
// stored: AutoNumber true, DBAccessibleFromOPCUA true, InstanceOfName FB21-Flush A, InstanceOfType FB
"FB21-Flush A"
BEGIN
END_DATA_BLOCK

DATA_BLOCK "FB23-regenarationpgmFB_DB"   // DB178
VERSION : 0.1
// stored: AutoNumber true, DBAccessibleFromOPCUA true, InstanceOfName FB23-regenarationpgmFB, InstanceOfType FB
"FB23-regenarationpgmFB"
BEGIN
END_DATA_BLOCK

DATA_BLOCK "FB3-Ratiocheck_DB"   // DB60
VERSION : 0.1
// stored: AutoNumber true, DBAccessibleFromOPCUA true, InstanceOfName FB3-Ratiocheck, InstanceOfType FB
"FB3-Ratiocheck"
BEGIN
END_DATA_BLOCK

DATA_BLOCK "FB5-Dearing with valveA_DB"   // DB4
VERSION : 0.1
// stored: AutoNumber true, DBAccessibleFromOPCUA true, InstanceOfName FB5-Dearing with valve, InstanceOfType FB
"FB5-Dearing with valve"
BEGIN
END_DATA_BLOCK

DATA_BLOCK "FB5-Dearing with valveB_DB"   // DB6
VERSION : 0.1
// stored: AutoNumber true, DBAccessibleFromOPCUA true, InstanceOfName FB5-Dearing with valve, InstanceOfType FB
"FB5-Dearing with valve"
BEGIN
END_DATA_BLOCK

DATA_BLOCK "LGF_FIFO_DB"   // DB285
AUTHOR : Siemens_Industry_Support
FAMILY : LGF
NAME : LGF_FIFO
VERSION : 0.1
// stored: AutoNumber true, DBAccessibleFromOPCUA true, InstanceOfName LGF_FIFO, InstanceOfType FB
"LGF_FIFO"
   // VAR_INPUT
   //    enqueue : Bool;
   //    dequeue : Bool;
   //    reset : Bool;
   //    clear : Bool;
   //    initialItem : Variant;
   // END_VAR
   // VAR_OUTPUT
   //    error { ExternalWritable := 'False'} : Bool;
   //    status { ExternalWritable := 'False'} : Word;
   //    subFunctionStatus { ExternalWritable := 'False'} : Word;
   //    elementCount { ExternalWritable := 'False'} : DInt;
   //    isEmpty { ExternalWritable := 'False'} : Bool;
   // END_VAR
   // VAR_IN_OUT
   //    item : Variant;
   //    buffer : Variant;
   // END_VAR
   // VAR
   //    statEdgesMem { ExternalAccessible := 'False'; ExternalVisible := 'False'; ExternalWritable := 'False'} : Struct
   //       enqueue { ExternalAccessible := 'False'; ExternalVisible := 'False'; ExternalWritable := 'False'} : Bool;
   //       dequeue { ExternalAccessible := 'False'; ExternalVisible := 'False'; ExternalWritable := 'False'} : Bool;
   //       clear { ExternalAccessible := 'False'; ExternalVisible := 'False'; ExternalWritable := 'False'} : Bool;
   //    END_STRUCT;
   //    statFirstItemIndex { ExternalAccessible := 'False'; ExternalVisible := 'False'; ExternalWritable := 'False'} : Int;
   //    statNextEmptyItemIndex { ExternalAccessible := 'False'; ExternalVisible := 'False'; ExternalWritable := 'False'} : Int;
   //    statElementCount { ExternalAccessible := 'False'; ExternalVisible := 'False'; ExternalWritable := 'False'} : DInt;
   // END_VAR
BEGIN
END_DATA_BLOCK

DATA_BLOCK "LGF_FIFO_DB_1"   // DB284
AUTHOR : Siemens_Industry_Support
FAMILY : LGF
NAME : LGF_FIFO
VERSION : 0.1
// stored: AutoNumber true, DBAccessibleFromOPCUA true, InstanceOfName LGF_FIFO, InstanceOfType FB
"LGF_FIFO"
   // VAR_INPUT
   //    enqueue : Bool;
   //    dequeue : Bool;
   //    reset : Bool;
   //    clear : Bool;
   //    initialItem : Variant;
   // END_VAR
   // VAR_OUTPUT
   //    error { ExternalWritable := 'False'} : Bool;
   //    status { ExternalWritable := 'False'} : Word;
   //    subFunctionStatus { ExternalWritable := 'False'} : Word;
   //    elementCount { ExternalWritable := 'False'} : DInt;
   //    isEmpty { ExternalWritable := 'False'} : Bool;
   // END_VAR
   // VAR_IN_OUT
   //    item : Variant;
   //    buffer : Variant;
   // END_VAR
   // VAR
   //    statEdgesMem { ExternalAccessible := 'False'; ExternalVisible := 'False'; ExternalWritable := 'False'} : Struct
   //       enqueue { ExternalAccessible := 'False'; ExternalVisible := 'False'; ExternalWritable := 'False'} : Bool;
   //       dequeue { ExternalAccessible := 'False'; ExternalVisible := 'False'; ExternalWritable := 'False'} : Bool;
   //       clear { ExternalAccessible := 'False'; ExternalVisible := 'False'; ExternalWritable := 'False'} : Bool;
   //    END_STRUCT;
   //    statFirstItemIndex { ExternalAccessible := 'False'; ExternalVisible := 'False'; ExternalWritable := 'False'} : Int;
   //    statNextEmptyItemIndex { ExternalAccessible := 'False'; ExternalVisible := 'False'; ExternalWritable := 'False'} : Int;
   //    statElementCount { ExternalAccessible := 'False'; ExternalVisible := 'False'; ExternalWritable := 'False'} : DInt;
   // END_VAR
BEGIN
END_DATA_BLOCK

DATA_BLOCK "MixingRatio_DB"   // DB137
VERSION : 0.1
// stored: AutoNumber true, DBAccessibleFromOPCUA true, InstanceOfName MixingRatio, InstanceOfType FB
"MixingRatio"
BEGIN
END_DATA_BLOCK

DATA_BLOCK "alm_DB"   // DB37
VERSION : 0.1
// stored: AutoNumber true, DBAccessibleFromOPCUA true, InstanceOfName alm, InstanceOfType FB
"alm"
BEGIN
END_DATA_BLOCK

DATA_BLOCK "hour_min_DB"   // DB27
VERSION : 0.1
// stored: AutoNumber true, DBAccessibleFromOPCUA true, InstanceOfName hour_min, InstanceOfType FB
"hour_min"
BEGIN
END_DATA_BLOCK

DATA_BLOCK "hour_min_DB_1"   // DB28
VERSION : 0.1
// stored: AutoNumber true, DBAccessibleFromOPCUA true, InstanceOfName hour_min, InstanceOfType FB
"hour_min"
BEGIN
END_DATA_BLOCK

DATA_BLOCK "hour_min_DB_2"   // DB29
VERSION : 0.1
// stored: AutoNumber true, DBAccessibleFromOPCUA true, InstanceOfName hour_min, InstanceOfType FB
"hour_min"
BEGIN
END_DATA_BLOCK

DATA_BLOCK "hour_min_DB_3"   // DB30
VERSION : 0.1
// stored: AutoNumber true, DBAccessibleFromOPCUA true, InstanceOfName hour_min, InstanceOfType FB
"hour_min"
BEGIN
END_DATA_BLOCK

DATA_BLOCK "FB10-heater_DB"   // DB11
VERSION : 0.1
// stored: AutoNumber true, DBAccessibleFromOPCUA true, InstanceOfName FB10-heater, InstanceOfType FB
"FB10-heater"
BEGIN
END_DATA_BLOCK

DATA_BLOCK "FB10-heater_DB_1"   // DB12
VERSION : 0.1
// stored: AutoNumber true, DBAccessibleFromOPCUA true, InstanceOfName FB10-heater, InstanceOfType FB
"FB10-heater"
BEGIN
END_DATA_BLOCK

DATA_BLOCK "FB10-heater_DB_2"   // DB13
VERSION : 0.1
// stored: AutoNumber true, DBAccessibleFromOPCUA true, InstanceOfName FB10-heater, InstanceOfType FB
"FB10-heater"
BEGIN
END_DATA_BLOCK

DATA_BLOCK "FB10-heater_DB_3"   // DB14
VERSION : 0.1
// stored: AutoNumber true, DBAccessibleFromOPCUA true, InstanceOfName FB10-heater, InstanceOfType FB
"FB10-heater"
BEGIN
END_DATA_BLOCK

DATA_BLOCK "FB23-IEC_Timer_0_DB"   // DB172
{ S7_Optimized_Access := 'TRUE' }
// stored: AutoNumber true, DBAccessibleFromOPCUA true, InstanceOfName IEC_TIMER, OfSystemLibElement IEC_TIMER, OfSystemLibVersion 1.0
"IEC_TIMER"
   // VAR
   //    PT : Time;
   //    ET { ExternalWritable := 'False'} : Time;
   //    IN : Bool;
   //    Q { ExternalWritable := 'False'} : Bool;
   // END_VAR
BEGIN
END_DATA_BLOCK

DATA_BLOCK "FB23-IEC_Timer_0_DB1"   // DB173
{ S7_Optimized_Access := 'TRUE' }
// stored: AutoNumber true, DBAccessibleFromOPCUA true, InstanceOfName IEC_TIMER, OfSystemLibElement IEC_TIMER, OfSystemLibVersion 1.0
"IEC_TIMER"
   // VAR
   //    PT : Time;
   //    ET { ExternalWritable := 'False'} : Time;
   //    IN : Bool;
   //    Q { ExternalWritable := 'False'} : Bool;
   // END_VAR
BEGIN
END_DATA_BLOCK

DATA_BLOCK "FB23-IEC_Timer_0_DB3"   // DB174
{ S7_Optimized_Access := 'TRUE' }
// stored: AutoNumber true, DBAccessibleFromOPCUA true, InstanceOfName IEC_TIMER, OfSystemLibElement IEC_TIMER, OfSystemLibVersion 1.0
"IEC_TIMER"
   // VAR
   //    PT : Time;
   //    ET { ExternalWritable := 'False'} : Time;
   //    IN : Bool;
   //    Q { ExternalWritable := 'False'} : Bool;
   // END_VAR
BEGIN
END_DATA_BLOCK

DATA_BLOCK "FB23-IEC_Timer_0_DB5"   // DB176
{ S7_Optimized_Access := 'TRUE' }
// stored: AutoNumber true, DBAccessibleFromOPCUA true, InstanceOfName IEC_TIMER, OfSystemLibElement IEC_TIMER, OfSystemLibVersion 1.0
"IEC_TIMER"
   // VAR
   //    PT : Time;
   //    ET { ExternalWritable := 'False'} : Time;
   //    IN : Bool;
   //    Q { ExternalWritable := 'False'} : Bool;
   // END_VAR
BEGIN
END_DATA_BLOCK

DATA_BLOCK "FB23-IEC_Timer_0_DB6"   // DB177
{ S7_Optimized_Access := 'TRUE' }
// stored: AutoNumber true, DBAccessibleFromOPCUA true, InstanceOfName IEC_TIMER, OfSystemLibElement IEC_TIMER, OfSystemLibVersion 1.0
"IEC_TIMER"
   // VAR
   //    PT : Time;
   //    ET { ExternalWritable := 'False'} : Time;
   //    IN : Bool;
   //    Q { ExternalWritable := 'False'} : Bool;
   // END_VAR
BEGIN
END_DATA_BLOCK

DATA_BLOCK "FB23-R_TRIG_DB1"   // DB170
// stored: AutoNumber true, DBAccessibleFromOPCUA true, InstanceOfName R_TRIG, OfSystemLibElement R_TRIG, OfSystemLibVersion 1.0
"R_TRIG"
   // VAR_INPUT
   //    CLK : Bool;
   // END_VAR
   // VAR_OUTPUT
   //    Q : Bool;
   // END_VAR
   // VAR
   //    Stat_Bit : Bool;
   // END_VAR
BEGIN
END_DATA_BLOCK

DATA_BLOCK "FB3-IEC_Timer_0_DB"   // DB16
{ S7_Optimized_Access := 'TRUE' }
// stored: AutoNumber true, DBAccessibleFromOPCUA true, InstanceOfName IEC_TIMER, OfSystemLibElement IEC_TIMER, OfSystemLibVersion 1.0
"IEC_TIMER"
   // VAR
   //    PT : Time;
   //    ET { ExternalWritable := 'False'} : Time;
   //    IN : Bool;
   //    Q { ExternalWritable := 'False'} : Bool;
   // END_VAR
BEGIN
END_DATA_BLOCK

DATA_BLOCK "FB3-IEC_Timer_0_DB1."   // DB17
{ S7_Optimized_Access := 'TRUE' }
// stored: AutoNumber true, DBAccessibleFromOPCUA true, InstanceOfName IEC_TIMER, OfSystemLibElement IEC_TIMER, OfSystemLibVersion 1.0
"IEC_TIMER"
   // VAR
   //    PT : Time;
   //    ET { ExternalWritable := 'False'} : Time;
   //    IN : Bool;
   //    Q { ExternalWritable := 'False'} : Bool;
   // END_VAR
BEGIN
END_DATA_BLOCK

DATA_BLOCK "FB3-IEC_Timer_0_DB3"   // DB19
{ S7_Optimized_Access := 'TRUE' }
// stored: AutoNumber true, DBAccessibleFromOPCUA true, InstanceOfName IEC_TIMER, OfSystemLibElement IEC_TIMER, OfSystemLibVersion 1.0
"IEC_TIMER"
   // VAR
   //    PT : Time;
   //    ET { ExternalWritable := 'False'} : Time;
   //    IN : Bool;
   //    Q { ExternalWritable := 'False'} : Bool;
   // END_VAR
BEGIN
END_DATA_BLOCK

DATA_BLOCK "FB3-IEC_Timer_0_DB4"   // DB20
{ S7_Optimized_Access := 'TRUE' }
// stored: AutoNumber true, DBAccessibleFromOPCUA true, InstanceOfName IEC_TIMER, OfSystemLibElement IEC_TIMER, OfSystemLibVersion 1.0
"IEC_TIMER"
   // VAR
   //    PT : Time;
   //    ET { ExternalWritable := 'False'} : Time;
   //    IN : Bool;
   //    Q { ExternalWritable := 'False'} : Bool;
   // END_VAR
BEGIN
END_DATA_BLOCK

DATA_BLOCK "FB3-IEC_Timer_0_DB6"   // DB22
{ S7_Optimized_Access := 'TRUE' }
// stored: AutoNumber true, DBAccessibleFromOPCUA true, InstanceOfName IEC_TIMER, OfSystemLibElement IEC_TIMER, OfSystemLibVersion 1.0
"IEC_TIMER"
   // VAR
   //    PT : Time;
   //    ET { ExternalWritable := 'False'} : Time;
   //    IN : Bool;
   //    Q { ExternalWritable := 'False'} : Bool;
   // END_VAR
BEGIN
END_DATA_BLOCK

DATA_BLOCK "FB3-R_TRIG_DB1"   // DB15
// stored: AutoNumber true, DBAccessibleFromOPCUA true, InstanceOfName R_TRIG, OfSystemLibElement R_TRIG, OfSystemLibVersion 1.0
"R_TRIG"
   // VAR_INPUT
   //    CLK : Bool;
   // END_VAR
   // VAR_OUTPUT
   //    Q : Bool;
   // END_VAR
   // VAR
   //    Stat_Bit : Bool;
   // END_VAR
BEGIN
END_DATA_BLOCK

DATA_BLOCK "F_TRIG_DB"   // DB86
// stored: AutoNumber true, DBAccessibleFromOPCUA true, InstanceOfName F_TRIG, OfSystemLibElement F_TRIG, OfSystemLibVersion 1.0
"F_TRIG"
   // VAR_INPUT
   //    CLK : Bool;
   // END_VAR
   // VAR_OUTPUT
   //    Q : Bool;
   // END_VAR
   // VAR
   //    Stat_Bit : Bool;
   // END_VAR
BEGIN
END_DATA_BLOCK

DATA_BLOCK "IEC_Counter_0_DB 10"   // DB304
{ S7_Optimized_Access := 'TRUE' }
// stored: AutoNumber true, DBAccessibleFromOPCUA true, InstanceOfName IEC_COUNTER, OfSystemLibElement IEC_COUNTER, OfSystemLibVersion 1.0
"IEC_COUNTER"
   // VAR RETAIN
   //    CU : Bool;
   //    CD : Bool;
   //    R : Bool;
   //    LD : Bool;
   //    QU : Bool;
   //    QD : Bool;
   //    PV : Int;
   //    CV : Int;
   // END_VAR
BEGIN
END_DATA_BLOCK

DATA_BLOCK "IEC_Counter_0_DB"   // DB139
{ S7_Optimized_Access := 'TRUE' }
// stored: AutoNumber true, DBAccessibleFromOPCUA true, InstanceOfName IEC_UDCOUNTER, OfSystemLibElement IEC_UDCOUNTER, OfSystemLibVersion 1.0
"IEC_UDCOUNTER"
   // VAR RETAIN
   //    CU : Bool;
   //    CD : Bool;
   //    R : Bool;
   //    LD : Bool;
   //    QU : Bool;
   //    QD : Bool;
   //    PV : UDInt;
   //    CV : UDInt;
   // END_VAR
BEGIN
END_DATA_BLOCK

DATA_BLOCK "IEC_Counter_0_DB_1"   // DB179
{ S7_Optimized_Access := 'TRUE' }
// stored: AutoNumber true, DBAccessibleFromOPCUA true, InstanceOfName IEC_COUNTER, OfSystemLibElement IEC_COUNTER, OfSystemLibVersion 1.0
"IEC_COUNTER"
   // VAR RETAIN
   //    CU : Bool;
   //    CD : Bool;
   //    R : Bool;
   //    LD : Bool;
   //    QU : Bool;
   //    QD : Bool;
   //    PV : Int;
   //    CV : Int;
   // END_VAR
BEGIN
END_DATA_BLOCK

DATA_BLOCK "IEC_Counter_0_DB_2"   // DB31
{ S7_Optimized_Access := 'TRUE' }
// stored: AutoNumber true, DBAccessibleFromOPCUA true, InstanceOfName IEC_UDCOUNTER, OfSystemLibElement IEC_UDCOUNTER, OfSystemLibVersion 1.0
"IEC_UDCOUNTER"
   // VAR RETAIN
   //    CU : Bool;
   //    CD : Bool;
   //    R : Bool;
   //    LD : Bool;
   //    QU : Bool;
   //    QD : Bool;
   //    PV : UDInt;
   //    CV : UDInt;
   // END_VAR
BEGIN
END_DATA_BLOCK

DATA_BLOCK "IEC_Timer_0_DB"   // DB9
{ S7_Optimized_Access := 'TRUE' }
// stored: AutoNumber true, DBAccessibleFromOPCUA true, InstanceOfName IEC_TIMER, OfSystemLibElement IEC_TIMER, OfSystemLibVersion 1.0
"IEC_TIMER"
   // VAR
   //    PT : Time;
   //    ET { ExternalWritable := 'False'} : Time;
   //    IN : Bool;
   //    Q { ExternalWritable := 'False'} : Bool;
   // END_VAR
BEGIN
END_DATA_BLOCK

DATA_BLOCK "IEC_Timer_0_DB_1"   // DB85
{ S7_Optimized_Access := 'TRUE' }
// stored: AutoNumber true, DBAccessibleFromOPCUA true, InstanceOfName IEC_TIMER, OfSystemLibElement IEC_TIMER, OfSystemLibVersion 1.0
"IEC_TIMER"
   // VAR
   //    PT : Time;
   //    ET { ExternalWritable := 'False'} : Time;
   //    IN : Bool;
   //    Q { ExternalWritable := 'False'} : Bool;
   // END_VAR
BEGIN
END_DATA_BLOCK

DATA_BLOCK "IEC_Timer_0_DB_10"   // DB69
{ S7_Optimized_Access := 'TRUE' }
// stored: AutoNumber true, DBAccessibleFromOPCUA true, InstanceOfName IEC_TIMER, OfSystemLibElement IEC_TIMER, OfSystemLibVersion 1.0
"IEC_TIMER"
   // VAR
   //    PT : Time;
   //    ET { ExternalWritable := 'False'} : Time;
   //    IN : Bool;
   //    Q { ExternalWritable := 'False'} : Bool;
   // END_VAR
BEGIN
END_DATA_BLOCK

DATA_BLOCK "IEC_Timer_0_DB_100"   // DB235
{ S7_Optimized_Access := 'TRUE' }
// stored: AutoNumber true, DBAccessibleFromOPCUA true, InstanceOfName IEC_TIMER, OfSystemLibElement IEC_TIMER, OfSystemLibVersion 1.0
"IEC_TIMER"
   // VAR
   //    PT : Time;
   //    ET { ExternalWritable := 'False'} : Time;
   //    IN : Bool;
   //    Q { ExternalWritable := 'False'} : Bool;
   // END_VAR
BEGIN
END_DATA_BLOCK

DATA_BLOCK "IEC_Timer_0_DB_101"   // DB236
{ S7_Optimized_Access := 'TRUE' }
// stored: AutoNumber true, DBAccessibleFromOPCUA true, InstanceOfName IEC_TIMER, OfSystemLibElement IEC_TIMER, OfSystemLibVersion 1.0
"IEC_TIMER"
   // VAR
   //    PT : Time;
   //    ET { ExternalWritable := 'False'} : Time;
   //    IN : Bool;
   //    Q { ExternalWritable := 'False'} : Bool;
   // END_VAR
BEGIN
END_DATA_BLOCK

DATA_BLOCK "IEC_Timer_0_DB_102"   // DB237
{ S7_Optimized_Access := 'TRUE' }
// stored: AutoNumber true, DBAccessibleFromOPCUA true, InstanceOfName IEC_TIMER, OfSystemLibElement IEC_TIMER, OfSystemLibVersion 1.0
"IEC_TIMER"
   // VAR
   //    PT : Time;
   //    ET { ExternalWritable := 'False'} : Time;
   //    IN : Bool;
   //    Q { ExternalWritable := 'False'} : Bool;
   // END_VAR
BEGIN
END_DATA_BLOCK

DATA_BLOCK "IEC_Timer_0_DB_106"   // DB242
{ S7_Optimized_Access := 'TRUE' }
// stored: AutoNumber true, DBAccessibleFromOPCUA true, InstanceOfName IEC_TIMER, OfSystemLibElement IEC_TIMER, OfSystemLibVersion 1.0
"IEC_TIMER"
   // VAR
   //    PT : Time;
   //    ET { ExternalWritable := 'False'} : Time;
   //    IN : Bool;
   //    Q { ExternalWritable := 'False'} : Bool;
   // END_VAR
BEGIN
END_DATA_BLOCK

DATA_BLOCK "IEC_Timer_0_DB_108"   // DB244
{ S7_Optimized_Access := 'TRUE' }
// stored: AutoNumber true, DBAccessibleFromOPCUA true, InstanceOfName IEC_TIMER, OfSystemLibElement IEC_TIMER, OfSystemLibVersion 1.0
"IEC_TIMER"
   // VAR
   //    PT : Time;
   //    ET { ExternalWritable := 'False'} : Time;
   //    IN : Bool;
   //    Q { ExternalWritable := 'False'} : Bool;
   // END_VAR
BEGIN
END_DATA_BLOCK

DATA_BLOCK "IEC_Timer_0_DB_11"   // DB8
{ S7_Optimized_Access := 'TRUE' }
// stored: AutoNumber true, DBAccessibleFromOPCUA true, InstanceOfName IEC_TIMER, OfSystemLibElement IEC_TIMER, OfSystemLibVersion 1.0
"IEC_TIMER"
   // VAR
   //    PT : Time;
   //    ET { ExternalWritable := 'False'} : Time;
   //    IN : Bool;
   //    Q { ExternalWritable := 'False'} : Bool;
   // END_VAR
BEGIN
END_DATA_BLOCK

DATA_BLOCK "IEC_Timer_0_DB_111"   // DB227
{ S7_Optimized_Access := 'TRUE' }
// stored: AutoNumber true, DBAccessibleFromOPCUA true, InstanceOfName IEC_TIMER, OfSystemLibElement IEC_TIMER, OfSystemLibVersion 1.0
"IEC_TIMER"
   // VAR
   //    PT : Time;
   //    ET { ExternalWritable := 'False'} : Time;
   //    IN : Bool;
   //    Q { ExternalWritable := 'False'} : Bool;
   // END_VAR
BEGIN
END_DATA_BLOCK

DATA_BLOCK "IEC_Timer_0_DB_118"   // DB171
{ S7_Optimized_Access := 'TRUE' }
// stored: AutoNumber true, DBAccessibleFromOPCUA true, InstanceOfName IEC_TIMER, OfSystemLibElement IEC_TIMER, OfSystemLibVersion 1.0
"IEC_TIMER"
   // VAR
   //    PT : Time;
   //    ET { ExternalWritable := 'False'} : Time;
   //    IN : Bool;
   //    Q { ExternalWritable := 'False'} : Bool;
   // END_VAR
BEGIN
END_DATA_BLOCK

DATA_BLOCK "IEC_Timer_0_DB_12"   // DB10
{ S7_Optimized_Access := 'TRUE' }
// stored: AutoNumber true, DBAccessibleFromOPCUA true, InstanceOfName IEC_TIMER, OfSystemLibElement IEC_TIMER, OfSystemLibVersion 1.0
"IEC_TIMER"
   // VAR
   //    PT : Time;
   //    ET { ExternalWritable := 'False'} : Time;
   //    IN : Bool;
   //    Q { ExternalWritable := 'False'} : Bool;
   // END_VAR
BEGIN
END_DATA_BLOCK

DATA_BLOCK "IEC_Timer_0_DB_120"   // DB224
{ S7_Optimized_Access := 'TRUE' }
// stored: AutoNumber true, DBAccessibleFromOPCUA true, InstanceOfName IEC_TIMER, OfSystemLibElement IEC_TIMER, OfSystemLibVersion 1.0
"IEC_TIMER"
   // VAR
   //    PT : Time;
   //    ET { ExternalWritable := 'False'} : Time;
   //    IN : Bool;
   //    Q { ExternalWritable := 'False'} : Bool;
   // END_VAR
BEGIN
END_DATA_BLOCK

DATA_BLOCK "IEC_Timer_0_DB_121"   // DB246
{ S7_Optimized_Access := 'TRUE' }
// stored: AutoNumber true, DBAccessibleFromOPCUA true, InstanceOfName IEC_TIMER, OfSystemLibElement IEC_TIMER, OfSystemLibVersion 1.0
"IEC_TIMER"
   // VAR
   //    PT : Time;
   //    ET { ExternalWritable := 'False'} : Time;
   //    IN : Bool;
   //    Q { ExternalWritable := 'False'} : Bool;
   // END_VAR
BEGIN
END_DATA_BLOCK

DATA_BLOCK "IEC_Timer_0_DB_122"   // DB247
{ S7_Optimized_Access := 'TRUE' }
// stored: AutoNumber true, DBAccessibleFromOPCUA true, InstanceOfName IEC_TIMER, OfSystemLibElement IEC_TIMER, OfSystemLibVersion 1.0
"IEC_TIMER"
   // VAR
   //    PT : Time;
   //    ET { ExternalWritable := 'False'} : Time;
   //    IN : Bool;
   //    Q { ExternalWritable := 'False'} : Bool;
   // END_VAR
BEGIN
END_DATA_BLOCK

DATA_BLOCK "IEC_Timer_0_DB_126"   // DB2
{ S7_Optimized_Access := 'TRUE' }
// stored: AutoNumber true, DBAccessibleFromOPCUA true, InstanceOfName IEC_TIMER, OfSystemLibElement IEC_TIMER, OfSystemLibVersion 1.0
"IEC_TIMER"
   // VAR
   //    PT : Time;
   //    ET { ExternalWritable := 'False'} : Time;
   //    IN : Bool;
   //    Q { ExternalWritable := 'False'} : Bool;
   // END_VAR
BEGIN
END_DATA_BLOCK

DATA_BLOCK "IEC_Timer_0_DB_127"   // DB3
{ S7_Optimized_Access := 'TRUE' }
// stored: AutoNumber true, DBAccessibleFromOPCUA true, InstanceOfName IEC_TIMER, OfSystemLibElement IEC_TIMER, OfSystemLibVersion 1.0
"IEC_TIMER"
   // VAR
   //    PT : Time;
   //    ET { ExternalWritable := 'False'} : Time;
   //    IN : Bool;
   //    Q { ExternalWritable := 'False'} : Bool;
   // END_VAR
BEGIN
END_DATA_BLOCK

DATA_BLOCK "IEC_Timer_0_DB_13"   // DB353
{ S7_Optimized_Access := 'TRUE' }
// stored: AutoNumber true, DBAccessibleFromOPCUA true, InstanceOfName IEC_TIMER, OfSystemLibElement IEC_TIMER, OfSystemLibVersion 1.0
"IEC_TIMER"
   // VAR
   //    PT : Time;
   //    ET { ExternalWritable := 'False'} : Time;
   //    IN : Bool;
   //    Q { ExternalWritable := 'False'} : Bool;
   // END_VAR
BEGIN
END_DATA_BLOCK

DATA_BLOCK "IEC_Timer_0_DB_14"   // DB33
{ S7_Optimized_Access := 'TRUE' }
// stored: AutoNumber true, DBAccessibleFromOPCUA true, InstanceOfName IEC_TIMER, OfSystemLibElement IEC_TIMER, OfSystemLibVersion 1.0
"IEC_TIMER"
   // VAR
   //    PT : Time;
   //    ET { ExternalWritable := 'False'} : Time;
   //    IN : Bool;
   //    Q { ExternalWritable := 'False'} : Bool;
   // END_VAR
BEGIN
END_DATA_BLOCK

DATA_BLOCK "IEC_Timer_0_DB_15"   // DB355
{ S7_Optimized_Access := 'TRUE' }
// stored: AutoNumber true, DBAccessibleFromOPCUA true, InstanceOfName IEC_TIMER, OfSystemLibElement IEC_TIMER, OfSystemLibVersion 1.0
"IEC_TIMER"
   // VAR
   //    PT : Time;
   //    ET { ExternalWritable := 'False'} : Time;
   //    IN : Bool;
   //    Q { ExternalWritable := 'False'} : Bool;
   // END_VAR
BEGIN
END_DATA_BLOCK

DATA_BLOCK "IEC_Timer_0_DB_16"   // DB34
{ S7_Optimized_Access := 'TRUE' }
// stored: AutoNumber true, DBAccessibleFromOPCUA true, InstanceOfName IEC_TIMER, OfSystemLibElement IEC_TIMER, OfSystemLibVersion 1.0
"IEC_TIMER"
   // VAR
   //    PT : Time;
   //    ET { ExternalWritable := 'False'} : Time;
   //    IN : Bool;
   //    Q { ExternalWritable := 'False'} : Bool;
   // END_VAR
BEGIN
END_DATA_BLOCK

DATA_BLOCK "IEC_Timer_0_DB_17"   // DB357
{ S7_Optimized_Access := 'TRUE' }
// stored: AutoNumber true, DBAccessibleFromOPCUA true, InstanceOfName IEC_TIMER, OfSystemLibElement IEC_TIMER, OfSystemLibVersion 1.0
"IEC_TIMER"
   // VAR
   //    PT : Time;
   //    ET { ExternalWritable := 'False'} : Time;
   //    IN : Bool;
   //    Q { ExternalWritable := 'False'} : Bool;
   // END_VAR
BEGIN
END_DATA_BLOCK

DATA_BLOCK "IEC_Timer_0_DB_18"   // DB35
{ S7_Optimized_Access := 'TRUE' }
// stored: AutoNumber true, DBAccessibleFromOPCUA true, InstanceOfName IEC_TIMER, OfSystemLibElement IEC_TIMER, OfSystemLibVersion 1.0
"IEC_TIMER"
   // VAR
   //    PT : Time;
   //    ET { ExternalWritable := 'False'} : Time;
   //    IN : Bool;
   //    Q { ExternalWritable := 'False'} : Bool;
   // END_VAR
BEGIN
END_DATA_BLOCK

DATA_BLOCK "IEC_Timer_0_DB_19"   // DB38
{ S7_Optimized_Access := 'TRUE' }
// stored: AutoNumber true, DBAccessibleFromOPCUA true, InstanceOfName IEC_TIMER, OfSystemLibElement IEC_TIMER, OfSystemLibVersion 1.0
"IEC_TIMER"
   // VAR
   //    PT : Time;
   //    ET { ExternalWritable := 'False'} : Time;
   //    IN : Bool;
   //    Q { ExternalWritable := 'False'} : Bool;
   // END_VAR
BEGIN
END_DATA_BLOCK

DATA_BLOCK "IEC_Timer_0_DB_2"   // DB166
{ S7_Optimized_Access := 'TRUE' }
// stored: AutoNumber true, DBAccessibleFromOPCUA true, InstanceOfName IEC_TIMER, OfSystemLibElement IEC_TIMER, OfSystemLibVersion 1.0
"IEC_TIMER"
   // VAR
   //    PT : Time;
   //    ET { ExternalWritable := 'False'} : Time;
   //    IN : Bool;
   //    Q { ExternalWritable := 'False'} : Bool;
   // END_VAR
BEGIN
END_DATA_BLOCK

DATA_BLOCK "IEC_Timer_0_DB_20"   // DB44
{ S7_Optimized_Access := 'TRUE' }
// stored: AutoNumber true, DBAccessibleFromOPCUA true, InstanceOfName IEC_TIMER, OfSystemLibElement IEC_TIMER, OfSystemLibVersion 1.0
"IEC_TIMER"
   // VAR
   //    PT : Time;
   //    ET { ExternalWritable := 'False'} : Time;
   //    IN : Bool;
   //    Q { ExternalWritable := 'False'} : Bool;
   // END_VAR
BEGIN
END_DATA_BLOCK

DATA_BLOCK "IEC_Timer_0_DB_21"   // DB50
{ S7_Optimized_Access := 'TRUE' }
// stored: AutoNumber true, DBAccessibleFromOPCUA true, InstanceOfName IEC_TIMER, OfSystemLibElement IEC_TIMER, OfSystemLibVersion 1.0
"IEC_TIMER"
   // VAR
   //    PT : Time;
   //    ET { ExternalWritable := 'False'} : Time;
   //    IN : Bool;
   //    Q { ExternalWritable := 'False'} : Bool;
   // END_VAR
BEGIN
END_DATA_BLOCK

DATA_BLOCK "IEC_Timer_0_DB_22"   // DB51
{ S7_Optimized_Access := 'TRUE' }
// stored: AutoNumber true, DBAccessibleFromOPCUA true, InstanceOfName IEC_TIMER, OfSystemLibElement IEC_TIMER, OfSystemLibVersion 1.0
"IEC_TIMER"
   // VAR
   //    PT : Time;
   //    ET { ExternalWritable := 'False'} : Time;
   //    IN : Bool;
   //    Q { ExternalWritable := 'False'} : Bool;
   // END_VAR
BEGIN
END_DATA_BLOCK

DATA_BLOCK "IEC_Timer_0_DB_23"   // DB53
{ S7_Optimized_Access := 'TRUE' }
// stored: AutoNumber true, DBAccessibleFromOPCUA true, InstanceOfName IEC_TIMER, OfSystemLibElement IEC_TIMER, OfSystemLibVersion 1.0
"IEC_TIMER"
   // VAR
   //    PT : Time;
   //    ET { ExternalWritable := 'False'} : Time;
   //    IN : Bool;
   //    Q { ExternalWritable := 'False'} : Bool;
   // END_VAR
BEGIN
END_DATA_BLOCK

DATA_BLOCK "IEC_Timer_0_DB_28"   // DB180
{ S7_Optimized_Access := 'TRUE' }
// stored: AutoNumber true, DBAccessibleFromOPCUA true, InstanceOfName IEC_TIMER, OfSystemLibElement IEC_TIMER, OfSystemLibVersion 1.0
"IEC_TIMER"
   // VAR
   //    PT : Time;
   //    ET { ExternalWritable := 'False'} : Time;
   //    IN : Bool;
   //    Q { ExternalWritable := 'False'} : Bool;
   // END_VAR
BEGIN
END_DATA_BLOCK

DATA_BLOCK "IEC_Timer_0_DB_3"   // DB117
{ S7_Optimized_Access := 'TRUE' }
// stored: AutoNumber true, DBAccessibleFromOPCUA true, InstanceOfName IEC_TIMER, OfSystemLibElement IEC_TIMER, OfSystemLibVersion 1.0
"IEC_TIMER"
   // VAR
   //    PT : Time;
   //    ET { ExternalWritable := 'False'} : Time;
   //    IN : Bool;
   //    Q { ExternalWritable := 'False'} : Bool;
   // END_VAR
BEGIN
END_DATA_BLOCK

DATA_BLOCK "IEC_Timer_0_DB_30"   // DB182
{ S7_Optimized_Access := 'TRUE' }
// stored: AutoNumber true, DBAccessibleFromOPCUA true, InstanceOfName IEC_TIMER, OfSystemLibElement IEC_TIMER, OfSystemLibVersion 1.0
"IEC_TIMER"
   // VAR
   //    PT : Time;
   //    ET { ExternalWritable := 'False'} : Time;
   //    IN : Bool;
   //    Q { ExternalWritable := 'False'} : Bool;
   // END_VAR
BEGIN
END_DATA_BLOCK

DATA_BLOCK "IEC_Timer_0_DB_31"   // DB183
{ S7_Optimized_Access := 'TRUE' }
// stored: AutoNumber true, DBAccessibleFromOPCUA true, InstanceOfName IEC_TIMER, OfSystemLibElement IEC_TIMER, OfSystemLibVersion 1.0
"IEC_TIMER"
   // VAR
   //    PT : Time;
   //    ET { ExternalWritable := 'False'} : Time;
   //    IN : Bool;
   //    Q { ExternalWritable := 'False'} : Bool;
   // END_VAR
BEGIN
END_DATA_BLOCK

DATA_BLOCK "IEC_Timer_0_DB_32"   // DB184
{ S7_Optimized_Access := 'TRUE' }
// stored: AutoNumber true, DBAccessibleFromOPCUA true, InstanceOfName IEC_TIMER, OfSystemLibElement IEC_TIMER, OfSystemLibVersion 1.0
"IEC_TIMER"
   // VAR
   //    PT : Time;
   //    ET { ExternalWritable := 'False'} : Time;
   //    IN : Bool;
   //    Q { ExternalWritable := 'False'} : Bool;
   // END_VAR
BEGIN
END_DATA_BLOCK

DATA_BLOCK "IEC_Timer_0_DB_33"   // DB275
{ S7_Optimized_Access := 'TRUE' }
// stored: AutoNumber true, DBAccessibleFromOPCUA true, InstanceOfName IEC_TIMER, OfSystemLibElement IEC_TIMER, OfSystemLibVersion 1.0
"IEC_TIMER"
   // VAR
   //    PT : Time;
   //    ET { ExternalWritable := 'False'} : Time;
   //    IN : Bool;
   //    Q { ExternalWritable := 'False'} : Bool;
   // END_VAR
BEGIN
END_DATA_BLOCK

DATA_BLOCK "IEC_Timer_0_DB_38"   // DB101
{ S7_Optimized_Access := 'TRUE' }
// stored: AutoNumber true, DBAccessibleFromOPCUA true, InstanceOfName IEC_TIMER, OfSystemLibElement IEC_TIMER, OfSystemLibVersion 1.0
"IEC_TIMER"
   // VAR
   //    PT : Time;
   //    ET { ExternalWritable := 'False'} : Time;
   //    IN : Bool;
   //    Q { ExternalWritable := 'False'} : Bool;
   // END_VAR
BEGIN
END_DATA_BLOCK

DATA_BLOCK "IEC_Timer_0_DB_39"   // DB346
{ S7_Optimized_Access := 'TRUE' }
// stored: AutoNumber true, DBAccessibleFromOPCUA true, InstanceOfName IEC_TIMER, OfSystemLibElement IEC_TIMER, OfSystemLibVersion 1.0
"IEC_TIMER"
   // VAR
   //    PT : Time;
   //    ET { ExternalWritable := 'False'} : Time;
   //    IN : Bool;
   //    Q { ExternalWritable := 'False'} : Bool;
   // END_VAR
BEGIN
END_DATA_BLOCK

DATA_BLOCK "IEC_Timer_0_DB_4"   // DB118
{ S7_Optimized_Access := 'TRUE' }
// stored: AutoNumber true, DBAccessibleFromOPCUA true, InstanceOfName IEC_TIMER, OfSystemLibElement IEC_TIMER, OfSystemLibVersion 1.0
"IEC_TIMER"
   // VAR
   //    PT : Time;
   //    ET { ExternalWritable := 'False'} : Time;
   //    IN : Bool;
   //    Q { ExternalWritable := 'False'} : Bool;
   // END_VAR
BEGIN
END_DATA_BLOCK

DATA_BLOCK "IEC_Timer_0_DB_40"   // DB347
{ S7_Optimized_Access := 'TRUE' }
// stored: AutoNumber true, DBAccessibleFromOPCUA true, InstanceOfName IEC_TIMER, OfSystemLibElement IEC_TIMER, OfSystemLibVersion 1.0
"IEC_TIMER"
   // VAR
   //    PT : Time;
   //    ET { ExternalWritable := 'False'} : Time;
   //    IN : Bool;
   //    Q { ExternalWritable := 'False'} : Bool;
   // END_VAR
BEGIN
END_DATA_BLOCK

DATA_BLOCK "IEC_Timer_0_DB_43"   // DB102
{ S7_Optimized_Access := 'TRUE' }
// stored: AutoNumber true, DBAccessibleFromOPCUA true, InstanceOfName IEC_TIMER, OfSystemLibElement IEC_TIMER, OfSystemLibVersion 1.0
"IEC_TIMER"
   // VAR
   //    PT : Time;
   //    ET { ExternalWritable := 'False'} : Time;
   //    IN : Bool;
   //    Q { ExternalWritable := 'False'} : Bool;
   // END_VAR
BEGIN
END_DATA_BLOCK

DATA_BLOCK "IEC_Timer_0_DB_48"   // DB313
{ S7_Optimized_Access := 'TRUE' }
// stored: AutoNumber true, DBAccessibleFromOPCUA true, InstanceOfName IEC_TIMER, OfSystemLibElement IEC_TIMER, OfSystemLibVersion 1.0
"IEC_TIMER"
   // VAR
   //    PT : Time;
   //    ET { ExternalWritable := 'False'} : Time;
   //    IN : Bool;
   //    Q { ExternalWritable := 'False'} : Bool;
   // END_VAR
BEGIN
END_DATA_BLOCK

DATA_BLOCK "IEC_Timer_0_DB_5"   // DB119
{ S7_Optimized_Access := 'TRUE' }
// stored: AutoNumber true, DBAccessibleFromOPCUA true, InstanceOfName IEC_TIMER, OfSystemLibElement IEC_TIMER, OfSystemLibVersion 1.0
"IEC_TIMER"
   // VAR
   //    PT : Time;
   //    ET { ExternalWritable := 'False'} : Time;
   //    IN : Bool;
   //    Q { ExternalWritable := 'False'} : Bool;
   // END_VAR
BEGIN
END_DATA_BLOCK

DATA_BLOCK "IEC_Timer_0_DB_53"   // DB305
{ S7_Optimized_Access := 'TRUE' }
// stored: AutoNumber true, DBAccessibleFromOPCUA true, InstanceOfName IEC_TIMER, OfSystemLibElement IEC_TIMER, OfSystemLibVersion 1.0
"IEC_TIMER"
   // VAR
   //    PT : Time;
   //    ET { ExternalWritable := 'False'} : Time;
   //    IN : Bool;
   //    Q { ExternalWritable := 'False'} : Bool;
   // END_VAR
BEGIN
END_DATA_BLOCK

DATA_BLOCK "IEC_Timer_0_DB_54"   // DB306
{ S7_Optimized_Access := 'TRUE' }
// stored: AutoNumber true, DBAccessibleFromOPCUA true, InstanceOfName IEC_TIMER, OfSystemLibElement IEC_TIMER, OfSystemLibVersion 1.0
"IEC_TIMER"
   // VAR
   //    PT : Time;
   //    ET { ExternalWritable := 'False'} : Time;
   //    IN : Bool;
   //    Q { ExternalWritable := 'False'} : Bool;
   // END_VAR
BEGIN
END_DATA_BLOCK

DATA_BLOCK "IEC_Timer_0_DB_55"   // DB308
{ S7_Optimized_Access := 'TRUE' }
// stored: AutoNumber true, DBAccessibleFromOPCUA true, InstanceOfName IEC_TIMER, OfSystemLibElement IEC_TIMER, OfSystemLibVersion 1.0
"IEC_TIMER"
   // VAR
   //    PT : Time;
   //    ET { ExternalWritable := 'False'} : Time;
   //    IN : Bool;
   //    Q { ExternalWritable := 'False'} : Bool;
   // END_VAR
BEGIN
END_DATA_BLOCK

DATA_BLOCK "IEC_Timer_0_DB_59"   // DB319
{ S7_Optimized_Access := 'TRUE' }
// stored: AutoNumber true, DBAccessibleFromOPCUA true, InstanceOfName IEC_TIMER, OfSystemLibElement IEC_TIMER, OfSystemLibVersion 1.0
"IEC_TIMER"
   // VAR
   //    PT : Time;
   //    ET { ExternalWritable := 'False'} : Time;
   //    IN : Bool;
   //    Q { ExternalWritable := 'False'} : Bool;
   // END_VAR
BEGIN
END_DATA_BLOCK

DATA_BLOCK "IEC_Timer_0_DB_6"   // DB120
{ S7_Optimized_Access := 'TRUE' }
// stored: AutoNumber true, DBAccessibleFromOPCUA true, InstanceOfName IEC_TIMER, OfSystemLibElement IEC_TIMER, OfSystemLibVersion 1.0
"IEC_TIMER"
   // VAR
   //    PT : Time;
   //    ET { ExternalWritable := 'False'} : Time;
   //    IN : Bool;
   //    Q { ExternalWritable := 'False'} : Bool;
   // END_VAR
BEGIN
END_DATA_BLOCK

DATA_BLOCK "IEC_Timer_0_DB_60"   // DB320
{ S7_Optimized_Access := 'TRUE' }
// stored: AutoNumber true, DBAccessibleFromOPCUA true, InstanceOfName IEC_TIMER, OfSystemLibElement IEC_TIMER, OfSystemLibVersion 1.0
"IEC_TIMER"
   // VAR
   //    PT : Time;
   //    ET { ExternalWritable := 'False'} : Time;
   //    IN : Bool;
   //    Q { ExternalWritable := 'False'} : Bool;
   // END_VAR
BEGIN
END_DATA_BLOCK

DATA_BLOCK "IEC_Timer_0_DB_7"   // DB168
{ S7_Optimized_Access := 'TRUE' }
// stored: AutoNumber true, DBAccessibleFromOPCUA true, InstanceOfName IEC_TIMER, OfSystemLibElement IEC_TIMER, OfSystemLibVersion 1.0
"IEC_TIMER"
   // VAR
   //    PT : Time;
   //    ET { ExternalWritable := 'False'} : Time;
   //    IN : Bool;
   //    Q { ExternalWritable := 'False'} : Bool;
   // END_VAR
BEGIN
END_DATA_BLOCK

DATA_BLOCK "IEC_Timer_0_DB_71"   // DB126
{ S7_Optimized_Access := 'TRUE' }
// stored: AutoNumber true, DBAccessibleFromOPCUA true, InstanceOfName IEC_TIMER, OfSystemLibElement IEC_TIMER, OfSystemLibVersion 1.0
"IEC_TIMER"
   // VAR
   //    PT : Time;
   //    ET { ExternalWritable := 'False'} : Time;
   //    IN : Bool;
   //    Q { ExternalWritable := 'False'} : Bool;
   // END_VAR
BEGIN
END_DATA_BLOCK

DATA_BLOCK "IEC_Timer_0_DB_72"   // DB129
{ S7_Optimized_Access := 'TRUE' }
// stored: AutoNumber true, DBAccessibleFromOPCUA true, InstanceOfName IEC_TIMER, OfSystemLibElement IEC_TIMER, OfSystemLibVersion 1.0
"IEC_TIMER"
   // VAR
   //    PT : Time;
   //    ET { ExternalWritable := 'False'} : Time;
   //    IN : Bool;
   //    Q { ExternalWritable := 'False'} : Bool;
   // END_VAR
BEGIN
END_DATA_BLOCK

DATA_BLOCK "IEC_Timer_0_DB_73"   // DB130
{ S7_Optimized_Access := 'TRUE' }
// stored: AutoNumber true, DBAccessibleFromOPCUA true, InstanceOfName IEC_TIMER, OfSystemLibElement IEC_TIMER, OfSystemLibVersion 1.0
"IEC_TIMER"
   // VAR
   //    PT : Time;
   //    ET { ExternalWritable := 'False'} : Time;
   //    IN : Bool;
   //    Q { ExternalWritable := 'False'} : Bool;
   // END_VAR
BEGIN
END_DATA_BLOCK

DATA_BLOCK "IEC_Timer_0_DB_74"   // DB131
{ S7_Optimized_Access := 'TRUE' }
// stored: AutoNumber true, DBAccessibleFromOPCUA true, InstanceOfName IEC_TIMER, OfSystemLibElement IEC_TIMER, OfSystemLibVersion 1.0
"IEC_TIMER"
   // VAR
   //    PT : Time;
   //    ET { ExternalWritable := 'False'} : Time;
   //    IN : Bool;
   //    Q { ExternalWritable := 'False'} : Bool;
   // END_VAR
BEGIN
END_DATA_BLOCK

DATA_BLOCK "IEC_Timer_0_DB_75"   // DB132
{ S7_Optimized_Access := 'TRUE' }
// stored: AutoNumber true, DBAccessibleFromOPCUA true, InstanceOfName IEC_TIMER, OfSystemLibElement IEC_TIMER, OfSystemLibVersion 1.0
"IEC_TIMER"
   // VAR
   //    PT : Time;
   //    ET { ExternalWritable := 'False'} : Time;
   //    IN : Bool;
   //    Q { ExternalWritable := 'False'} : Bool;
   // END_VAR
BEGIN
END_DATA_BLOCK

DATA_BLOCK "IEC_Timer_0_DB_76"   // DB133
{ S7_Optimized_Access := 'TRUE' }
// stored: AutoNumber true, DBAccessibleFromOPCUA true, InstanceOfName IEC_TIMER, OfSystemLibElement IEC_TIMER, OfSystemLibVersion 1.0
"IEC_TIMER"
   // VAR
   //    PT : Time;
   //    ET { ExternalWritable := 'False'} : Time;
   //    IN : Bool;
   //    Q { ExternalWritable := 'False'} : Bool;
   // END_VAR
BEGIN
END_DATA_BLOCK

DATA_BLOCK "IEC_Timer_0_DB_8"   // DB21
{ S7_Optimized_Access := 'TRUE' }
// stored: AutoNumber true, DBAccessibleFromOPCUA true, InstanceOfName IEC_TIMER, OfSystemLibElement IEC_TIMER, OfSystemLibVersion 1.0
"IEC_TIMER"
   // VAR
   //    PT : Time;
   //    ET { ExternalWritable := 'False'} : Time;
   //    IN : Bool;
   //    Q { ExternalWritable := 'False'} : Bool;
   // END_VAR
BEGIN
END_DATA_BLOCK

DATA_BLOCK "IEC_Timer_0_DB_81"   // DB219
{ S7_Optimized_Access := 'TRUE' }
// stored: AutoNumber true, DBAccessibleFromOPCUA true, InstanceOfName IEC_TIMER, OfSystemLibElement IEC_TIMER, OfSystemLibVersion 1.0
"IEC_TIMER"
   // VAR
   //    PT : Time;
   //    ET { ExternalWritable := 'False'} : Time;
   //    IN : Bool;
   //    Q { ExternalWritable := 'False'} : Bool;
   // END_VAR
BEGIN
END_DATA_BLOCK

DATA_BLOCK "IEC_Timer_0_DB_86"   // DB144
{ S7_Optimized_Access := 'TRUE' }
// stored: AutoNumber true, DBAccessibleFromOPCUA true, InstanceOfName IEC_TIMER, OfSystemLibElement IEC_TIMER, OfSystemLibVersion 1.0
"IEC_TIMER"
   // VAR
   //    PT : Time;
   //    ET { ExternalWritable := 'False'} : Time;
   //    IN : Bool;
   //    Q { ExternalWritable := 'False'} : Bool;
   // END_VAR
BEGIN
END_DATA_BLOCK

DATA_BLOCK "IEC_Timer_0_DB_87"   // DB207
{ S7_Optimized_Access := 'TRUE' }
// stored: AutoNumber true, DBAccessibleFromOPCUA true, InstanceOfName IEC_TIMER, OfSystemLibElement IEC_TIMER, OfSystemLibVersion 1.0
"IEC_TIMER"
   // VAR
   //    PT : Time;
   //    ET { ExternalWritable := 'False'} : Time;
   //    IN : Bool;
   //    Q { ExternalWritable := 'False'} : Bool;
   // END_VAR
BEGIN
END_DATA_BLOCK

DATA_BLOCK "IEC_Timer_0_DB_88"   // DB209
{ S7_Optimized_Access := 'TRUE' }
// stored: AutoNumber true, DBAccessibleFromOPCUA true, InstanceOfName IEC_TIMER, OfSystemLibElement IEC_TIMER, OfSystemLibVersion 1.0
"IEC_TIMER"
   // VAR
   //    PT : Time;
   //    ET { ExternalWritable := 'False'} : Time;
   //    IN : Bool;
   //    Q { ExternalWritable := 'False'} : Bool;
   // END_VAR
BEGIN
END_DATA_BLOCK

DATA_BLOCK "IEC_Timer_0_DB_89"   // DB210
{ S7_Optimized_Access := 'TRUE' }
// stored: AutoNumber true, DBAccessibleFromOPCUA true, InstanceOfName IEC_TIMER, OfSystemLibElement IEC_TIMER, OfSystemLibVersion 1.0
"IEC_TIMER"
   // VAR
   //    PT : Time;
   //    ET { ExternalWritable := 'False'} : Time;
   //    IN : Bool;
   //    Q { ExternalWritable := 'False'} : Bool;
   // END_VAR
BEGIN
END_DATA_BLOCK

DATA_BLOCK "IEC_Timer_0_DB_9"   // DB32
{ S7_Optimized_Access := 'TRUE' }
// stored: AutoNumber true, DBAccessibleFromOPCUA true, InstanceOfName IEC_TIMER, OfSystemLibElement IEC_TIMER, OfSystemLibVersion 1.0
"IEC_TIMER"
   // VAR
   //    PT : Time;
   //    ET { ExternalWritable := 'False'} : Time;
   //    IN : Bool;
   //    Q { ExternalWritable := 'False'} : Bool;
   // END_VAR
BEGIN
END_DATA_BLOCK

DATA_BLOCK "IEC_Timer_0_DB_90"   // DB211
{ S7_Optimized_Access := 'TRUE' }
// stored: AutoNumber true, DBAccessibleFromOPCUA true, InstanceOfName IEC_TIMER, OfSystemLibElement IEC_TIMER, OfSystemLibVersion 1.0
"IEC_TIMER"
   // VAR
   //    PT : Time;
   //    ET { ExternalWritable := 'False'} : Time;
   //    IN : Bool;
   //    Q { ExternalWritable := 'False'} : Bool;
   // END_VAR
BEGIN
END_DATA_BLOCK

DATA_BLOCK "IEC_Timer_0_DB_91"   // DB212
{ S7_Optimized_Access := 'TRUE' }
// stored: AutoNumber true, DBAccessibleFromOPCUA true, InstanceOfName IEC_TIMER, OfSystemLibElement IEC_TIMER, OfSystemLibVersion 1.0
"IEC_TIMER"
   // VAR
   //    PT : Time;
   //    ET { ExternalWritable := 'False'} : Time;
   //    IN : Bool;
   //    Q { ExternalWritable := 'False'} : Bool;
   // END_VAR
BEGIN
END_DATA_BLOCK

DATA_BLOCK "IEC_Timer_0_DB_92"   // DB213
{ S7_Optimized_Access := 'TRUE' }
// stored: AutoNumber true, DBAccessibleFromOPCUA true, InstanceOfName IEC_TIMER, OfSystemLibElement IEC_TIMER, OfSystemLibVersion 1.0
"IEC_TIMER"
   // VAR
   //    PT : Time;
   //    ET { ExternalWritable := 'False'} : Time;
   //    IN : Bool;
   //    Q { ExternalWritable := 'False'} : Bool;
   // END_VAR
BEGIN
END_DATA_BLOCK

DATA_BLOCK "IEC_Timer_0_DB_93"   // DB214
{ S7_Optimized_Access := 'TRUE' }
// stored: AutoNumber true, DBAccessibleFromOPCUA true, InstanceOfName IEC_TIMER, OfSystemLibElement IEC_TIMER, OfSystemLibVersion 1.0
"IEC_TIMER"
   // VAR
   //    PT : Time;
   //    ET { ExternalWritable := 'False'} : Time;
   //    IN : Bool;
   //    Q { ExternalWritable := 'False'} : Bool;
   // END_VAR
BEGIN
END_DATA_BLOCK

DATA_BLOCK "IEC_Timer_0_DB_94"   // DB215
{ S7_Optimized_Access := 'TRUE' }
// stored: AutoNumber true, DBAccessibleFromOPCUA true, InstanceOfName IEC_TIMER, OfSystemLibElement IEC_TIMER, OfSystemLibVersion 1.0
"IEC_TIMER"
   // VAR
   //    PT : Time;
   //    ET { ExternalWritable := 'False'} : Time;
   //    IN : Bool;
   //    Q { ExternalWritable := 'False'} : Bool;
   // END_VAR
BEGIN
END_DATA_BLOCK

DATA_BLOCK "IEC_Timer_0_DB_98"   // DB229
{ S7_Optimized_Access := 'TRUE' }
// stored: AutoNumber true, DBAccessibleFromOPCUA true, InstanceOfName IEC_TIMER, OfSystemLibElement IEC_TIMER, OfSystemLibVersion 1.0
"IEC_TIMER"
   // VAR
   //    PT : Time;
   //    ET { ExternalWritable := 'False'} : Time;
   //    IN : Bool;
   //    Q { ExternalWritable := 'False'} : Bool;
   // END_VAR
BEGIN
END_DATA_BLOCK

DATA_BLOCK "R_TRIG_DB"   // DB226
// stored: AutoNumber true, DBAccessibleFromOPCUA true, InstanceOfName R_TRIG, OfSystemLibElement R_TRIG, OfSystemLibVersion 1.0
"R_TRIG"
   // VAR_INPUT
   //    CLK : Bool;
   // END_VAR
   // VAR_OUTPUT
   //    Q : Bool;
   // END_VAR
   // VAR
   //    Stat_Bit : Bool;
   // END_VAR
BEGIN
END_DATA_BLOCK

DATA_BLOCK "R_TRIG_DB_1"   // DB23
// stored: AutoNumber true, DBAccessibleFromOPCUA true, InstanceOfName R_TRIG, OfSystemLibElement R_TRIG, OfSystemLibVersion 1.0
"R_TRIG"
   // VAR_INPUT
   //    CLK : Bool;
   // END_VAR
   // VAR_OUTPUT
   //    Q : Bool;
   // END_VAR
   // VAR
   //    Stat_Bit : Bool;
   // END_VAR
BEGIN
END_DATA_BLOCK

DATA_BLOCK "R_TRIG_DB_10"   // DB194
// stored: AutoNumber true, DBAccessibleFromOPCUA true, InstanceOfName R_TRIG, OfSystemLibElement R_TRIG, OfSystemLibVersion 1.0
"R_TRIG"
   // VAR_INPUT
   //    CLK : Bool;
   // END_VAR
   // VAR_OUTPUT
   //    Q : Bool;
   // END_VAR
   // VAR
   //    Stat_Bit : Bool;
   // END_VAR
BEGIN
END_DATA_BLOCK

DATA_BLOCK "R_TRIG_DB_11"   // DB195
// stored: AutoNumber true, DBAccessibleFromOPCUA true, InstanceOfName R_TRIG, OfSystemLibElement R_TRIG, OfSystemLibVersion 1.0
"R_TRIG"
   // VAR_INPUT
   //    CLK : Bool;
   // END_VAR
   // VAR_OUTPUT
   //    Q : Bool;
   // END_VAR
   // VAR
   //    Stat_Bit : Bool;
   // END_VAR
BEGIN
END_DATA_BLOCK

DATA_BLOCK "R_TRIG_DB_12"   // DB196
// stored: AutoNumber true, DBAccessibleFromOPCUA true, InstanceOfName R_TRIG, OfSystemLibElement R_TRIG, OfSystemLibVersion 1.0
"R_TRIG"
   // VAR_INPUT
   //    CLK : Bool;
   // END_VAR
   // VAR_OUTPUT
   //    Q : Bool;
   // END_VAR
   // VAR
   //    Stat_Bit : Bool;
   // END_VAR
BEGIN
END_DATA_BLOCK

DATA_BLOCK "R_TRIG_DB_13"   // DB197
// stored: AutoNumber true, DBAccessibleFromOPCUA true, InstanceOfName R_TRIG, OfSystemLibElement R_TRIG, OfSystemLibVersion 1.0
"R_TRIG"
   // VAR_INPUT
   //    CLK : Bool;
   // END_VAR
   // VAR_OUTPUT
   //    Q : Bool;
   // END_VAR
   // VAR
   //    Stat_Bit : Bool;
   // END_VAR
BEGIN
END_DATA_BLOCK

DATA_BLOCK "R_TRIG_DB_14"   // DB198
// stored: AutoNumber true, DBAccessibleFromOPCUA true, InstanceOfName R_TRIG, OfSystemLibElement R_TRIG, OfSystemLibVersion 1.0
"R_TRIG"
   // VAR_INPUT
   //    CLK : Bool;
   // END_VAR
   // VAR_OUTPUT
   //    Q : Bool;
   // END_VAR
   // VAR
   //    Stat_Bit : Bool;
   // END_VAR
BEGIN
END_DATA_BLOCK

DATA_BLOCK "R_TRIG_DB_15"   // DB199
// stored: AutoNumber true, DBAccessibleFromOPCUA true, InstanceOfName R_TRIG, OfSystemLibElement R_TRIG, OfSystemLibVersion 1.0
"R_TRIG"
   // VAR_INPUT
   //    CLK : Bool;
   // END_VAR
   // VAR_OUTPUT
   //    Q : Bool;
   // END_VAR
   // VAR
   //    Stat_Bit : Bool;
   // END_VAR
BEGIN
END_DATA_BLOCK

DATA_BLOCK "R_TRIG_DB_16"   // DB265
// stored: AutoNumber true, DBAccessibleFromOPCUA true, InstanceOfName R_TRIG, OfSystemLibElement R_TRIG, OfSystemLibVersion 1.0
"R_TRIG"
   // VAR_INPUT
   //    CLK : Bool;
   // END_VAR
   // VAR_OUTPUT
   //    Q : Bool;
   // END_VAR
   // VAR
   //    Stat_Bit : Bool;
   // END_VAR
BEGIN
END_DATA_BLOCK

DATA_BLOCK "R_TRIG_DB_17"   // DB333
// stored: AutoNumber true, DBAccessibleFromOPCUA true, InstanceOfName R_TRIG, OfSystemLibElement R_TRIG, OfSystemLibVersion 1.0
"R_TRIG"
   // VAR_INPUT
   //    CLK : Bool;
   // END_VAR
   // VAR_OUTPUT
   //    Q : Bool;
   // END_VAR
   // VAR
   //    Stat_Bit : Bool;
   // END_VAR
BEGIN
END_DATA_BLOCK

DATA_BLOCK "R_TRIG_DB_18"   // DB240
// stored: AutoNumber true, DBAccessibleFromOPCUA true, InstanceOfName R_TRIG, OfSystemLibElement R_TRIG, OfSystemLibVersion 1.0
"R_TRIG"
   // VAR_INPUT
   //    CLK : Bool;
   // END_VAR
   // VAR_OUTPUT
   //    Q : Bool;
   // END_VAR
   // VAR
   //    Stat_Bit : Bool;
   // END_VAR
BEGIN
END_DATA_BLOCK

DATA_BLOCK "R_TRIG_DB_19"   // DB332
// stored: AutoNumber true, DBAccessibleFromOPCUA true, InstanceOfName R_TRIG, OfSystemLibElement R_TRIG, OfSystemLibVersion 1.0
"R_TRIG"
   // VAR_INPUT
   //    CLK : Bool;
   // END_VAR
   // VAR_OUTPUT
   //    Q : Bool;
   // END_VAR
   // VAR
   //    Stat_Bit : Bool;
   // END_VAR
BEGIN
END_DATA_BLOCK

DATA_BLOCK "R_TRIG_DB_2"   // DB186
// stored: AutoNumber true, DBAccessibleFromOPCUA true, InstanceOfName R_TRIG, OfSystemLibElement R_TRIG, OfSystemLibVersion 1.0
"R_TRIG"
   // VAR_INPUT
   //    CLK : Bool;
   // END_VAR
   // VAR_OUTPUT
   //    Q : Bool;
   // END_VAR
   // VAR
   //    Stat_Bit : Bool;
   // END_VAR
BEGIN
END_DATA_BLOCK

DATA_BLOCK "R_TRIG_DB_20"   // DB231
// stored: AutoNumber true, DBAccessibleFromOPCUA true, InstanceOfName R_TRIG, OfSystemLibElement R_TRIG, OfSystemLibVersion 1.0
"R_TRIG"
   // VAR_INPUT
   //    CLK : Bool;
   // END_VAR
   // VAR_OUTPUT
   //    Q : Bool;
   // END_VAR
   // VAR
   //    Stat_Bit : Bool;
   // END_VAR
BEGIN
END_DATA_BLOCK

DATA_BLOCK "R_TRIG_DB_21"   // DB25
// stored: AutoNumber true, DBAccessibleFromOPCUA true, InstanceOfName R_TRIG, OfSystemLibElement R_TRIG, OfSystemLibVersion 1.0
"R_TRIG"
   // VAR_INPUT
   //    CLK : Bool;
   // END_VAR
   // VAR_OUTPUT
   //    Q : Bool;
   // END_VAR
   // VAR
   //    Stat_Bit : Bool;
   // END_VAR
BEGIN
END_DATA_BLOCK

DATA_BLOCK "R_TRIG_DB_23"   // DB309
// stored: AutoNumber true, DBAccessibleFromOPCUA true, InstanceOfName R_TRIG, OfSystemLibElement R_TRIG, OfSystemLibVersion 1.0
"R_TRIG"
   // VAR_INPUT
   //    CLK : Bool;
   // END_VAR
   // VAR_OUTPUT
   //    Q : Bool;
   // END_VAR
   // VAR
   //    Stat_Bit : Bool;
   // END_VAR
BEGIN
END_DATA_BLOCK

DATA_BLOCK "R_TRIG_DB_24"   // DB310
// stored: AutoNumber true, DBAccessibleFromOPCUA true, InstanceOfName R_TRIG, OfSystemLibElement R_TRIG, OfSystemLibVersion 1.0
"R_TRIG"
   // VAR_INPUT
   //    CLK : Bool;
   // END_VAR
   // VAR_OUTPUT
   //    Q : Bool;
   // END_VAR
   // VAR
   //    Stat_Bit : Bool;
   // END_VAR
BEGIN
END_DATA_BLOCK

DATA_BLOCK "R_TRIG_DB_3"   // DB187
// stored: AutoNumber true, DBAccessibleFromOPCUA true, InstanceOfName R_TRIG, OfSystemLibElement R_TRIG, OfSystemLibVersion 1.0
"R_TRIG"
   // VAR_INPUT
   //    CLK : Bool;
   // END_VAR
   // VAR_OUTPUT
   //    Q : Bool;
   // END_VAR
   // VAR
   //    Stat_Bit : Bool;
   // END_VAR
BEGIN
END_DATA_BLOCK

DATA_BLOCK "R_TRIG_DB_4"   // DB188
// stored: AutoNumber true, DBAccessibleFromOPCUA true, InstanceOfName R_TRIG, OfSystemLibElement R_TRIG, OfSystemLibVersion 1.0
"R_TRIG"
   // VAR_INPUT
   //    CLK : Bool;
   // END_VAR
   // VAR_OUTPUT
   //    Q : Bool;
   // END_VAR
   // VAR
   //    Stat_Bit : Bool;
   // END_VAR
BEGIN
END_DATA_BLOCK

DATA_BLOCK "R_TRIG_DB_5"   // DB189
// stored: AutoNumber true, DBAccessibleFromOPCUA true, InstanceOfName R_TRIG, OfSystemLibElement R_TRIG, OfSystemLibVersion 1.0
"R_TRIG"
   // VAR_INPUT
   //    CLK : Bool;
   // END_VAR
   // VAR_OUTPUT
   //    Q : Bool;
   // END_VAR
   // VAR
   //    Stat_Bit : Bool;
   // END_VAR
BEGIN
END_DATA_BLOCK

DATA_BLOCK "R_TRIG_DB_6"   // DB190
// stored: AutoNumber true, DBAccessibleFromOPCUA true, InstanceOfName R_TRIG, OfSystemLibElement R_TRIG, OfSystemLibVersion 1.0
"R_TRIG"
   // VAR_INPUT
   //    CLK : Bool;
   // END_VAR
   // VAR_OUTPUT
   //    Q : Bool;
   // END_VAR
   // VAR
   //    Stat_Bit : Bool;
   // END_VAR
BEGIN
END_DATA_BLOCK

DATA_BLOCK "R_TRIG_DB_7"   // DB191
// stored: AutoNumber true, DBAccessibleFromOPCUA true, InstanceOfName R_TRIG, OfSystemLibElement R_TRIG, OfSystemLibVersion 1.0
"R_TRIG"
   // VAR_INPUT
   //    CLK : Bool;
   // END_VAR
   // VAR_OUTPUT
   //    Q : Bool;
   // END_VAR
   // VAR
   //    Stat_Bit : Bool;
   // END_VAR
BEGIN
END_DATA_BLOCK

DATA_BLOCK "R_TRIG_DB_8"   // DB192
// stored: AutoNumber true, DBAccessibleFromOPCUA true, InstanceOfName R_TRIG, OfSystemLibElement R_TRIG, OfSystemLibVersion 1.0
"R_TRIG"
   // VAR_INPUT
   //    CLK : Bool;
   // END_VAR
   // VAR_OUTPUT
   //    Q : Bool;
   // END_VAR
   // VAR
   //    Stat_Bit : Bool;
   // END_VAR
BEGIN
END_DATA_BLOCK

DATA_BLOCK "R_TRIG_DB_9"   // DB193
// stored: AutoNumber true, DBAccessibleFromOPCUA true, InstanceOfName R_TRIG, OfSystemLibElement R_TRIG, OfSystemLibVersion 1.0
"R_TRIG"
   // VAR_INPUT
   //    CLK : Bool;
   // END_VAR
   // VAR_OUTPUT
   //    Q : Bool;
   // END_VAR
   // VAR
   //    Stat_Bit : Bool;
   // END_VAR
BEGIN
END_DATA_BLOCK
